   1:  PR[GP1:91,2] = PR[GP1:90,2] + -14.503;
   1:L PR[91] R[100]mm/sec CNT100;
   1:  PR[GP1:91,1] = PR[GP1:90,1] + -1.505;
   1:  PR[GP1:91,2] = PR[GP1:90,2] + -14.417;
   1:L PR[91] R[100]mm/sec CNT100;
   1:  PR[GP1:91,1] = PR[GP1:90,1] + -1.291;
   1:  PR[GP1:91,2] = PR[GP1:90,2] + -14.246;
   1:L PR[91] R[100]mm/sec CNT100;
   1:  PR[GP1:91,1] = PR[GP1:90,1] + -0.380;
   1:  PR[GP1:91,2] = PR[GP1:90,2] + -13.601;
   1:L PR[91] R[100]mm/sec CNT100;
   1:  PR[GP1:91,1] = PR[GP1:90,1] + 1.422;
   1:  PR[GP1:91,2] = PR[GP1:90,2] + -14.238;
   1:L PR[91] R[100]mm/sec CNT100;
   1:  PR[GP1:91,1] = PR[GP1:90,1] + 2.035;
   1:  PR[GP1:91,2] = PR[GP1:90,2] + -14.610;
   1:L PR[91] R[100]mm/sec CNT100;
   1:  PR[GP1:91,1] = PR[GP1:90,1] + 3.752;
   1:  PR[GP1:91,2] = PR[GP1:90,2] + -16.116;
   1:L PR[91] R[100]mm/sec CNT100;
   1:  PR[GP1:91,1] = PR[GP1:90,1] + 4.817;
   1:  PR[GP1:91,2] = PR[GP1:90,2] + -16.798;
   1:L PR[91] R[100]mm/sec CNT100;
   1:  PR[GP1:91,1] = PR[GP1:90,1] + 5.963;
   1:  PR[GP1:91,2] = PR[GP1:90,2] + -17.587;
   1:L PR[91] R[100]mm/sec CNT100;
   1:  PR[GP1:91,1] = PR[GP1:90,1] + 7.771;
   1:  PR[GP1:91,2] = PR[GP1:90,2] + -18.377;
   1:L PR[91] R[100]mm/sec CNT100;
   1:  PR[GP1:91,1] = PR[GP1:90,1] + 10.090;
   1:  PR[GP1:91,2] = PR[GP1:90,2] + -19.365;
   1:L PR[91] R[100]mm/sec CNT100;
   1:  PR[GP1:91,1] = PR[GP1:90,1] + 12.101;
   1:  PR[GP1:91,2] = PR[GP1:90,2] + -19.886;
   1:L PR[91] R[100]mm/sec CNT100;
   1:  PR[GP1:91,1] = PR[GP1:90,1] + 14.567;
   1:  PR[GP1:91,2] = PR[GP1:90,2] + -20.145;
   1:L PR[91] R[100]mm/sec CNT100;
   1:  PR[GP1:91,1] = PR[GP1:90,1] + 16.414;
   1:  PR[GP1:91,2] = PR[GP1:90,2] + -20.401;
   1:L PR[91] R[100]mm/sec CNT100;
   1:  PR[GP1:91,1] = PR[GP1:90,1] + 18.916;
   1:  PR[GP1:91,2] = PR[GP1:90,2] + -20.272;
   1:L PR[91] R[100]mm/sec CNT100;
   1:  PR[GP1:91,1] = PR[GP1:90,1] + 20.354;
   1:  PR[GP1:91,2] = PR[GP1:90,2] + -20.104;
   1:L PR[91] R[100]mm/sec CNT100;
   1:  PR[GP1:91,1] = PR[GP1:90,1] + 22.923;
   1:  PR[GP1:91,2] = PR[GP1:90,2] + -19.572;
   1:L PR[91] R[100]mm/sec CNT100;
   1:  PR[GP1:91,1] = PR[GP1:90,1] + 25.749;
   1:  PR[GP1:91,2] = PR[GP1:90,2] + -18.528;
   1:L PR[91] R[100]mm/sec CNT100;
   1:  PR[GP1:91,1] = PR[GP1:90,1] + 26.499;
   1:  PR[GP1:91,2] = PR[GP1:90,2] + -18.236;
   1:L PR[91] R[100]mm/sec CNT100;
   1:  PR[GP1:91,1] = PR[GP1:90,1] + 29.104;
   1:  PR[GP1:91,2] = PR[GP1:90,2] + -16.785;
   1:L PR[91] R[100]mm/sec CNT100;
   1:  PR[GP1:91,1] = PR[GP1:90,1] + 31.898;
   1:  PR[GP1:91,2] = PR[GP1:90,2] + -14.631;
   1:L PR[91] R[100]mm/sec CNT100;
   1:  PR[GP1:91,1] = PR[GP1:90,1] + 34.116;
   1:  PR[GP1:91,2] = PR[GP1:90,2] + -12.234;
   1:L PR[91] R[100]mm/sec CNT100;
   1:  PR[GP1:91,1] = PR[GP1:90,1] + 35.935;
   1:  PR[GP1:91,2] = PR[GP1:90,2] + -9.483;
   1:L PR[91] R[100]mm/sec CNT100;
   1:  PR[GP1:91,1] = PR[GP1:90,1] + 37.166;
   1:  PR[GP1:91,2] = PR[GP1:90,2] + -6.758;
   1:L PR[91] R[100]mm/sec CNT100;
   1:  PR[GP1:91,1] = PR[GP1:90,1] + 37.334;
   1:  PR[GP1:91,2] = PR[GP1:90,2] + -6.340;
   1:L PR[91] R[100]mm/sec CNT100;
   1:  PR[GP1:91,1] = PR[GP1:90,1] + 38.017;
   1:  PR[GP1:91,2] = PR[GP1:90,2] + -3.738;
   1:L PR[91] R[100]mm/sec CNT100;
   1:  PR[GP1:91,1] = PR[GP1:90,1] + 38.097;
   1:  PR[GP1:91,2] = PR[GP1:90,2] + -3.101;
   1:L PR[91] R[100]mm/sec CNT100;
   1:  PR[GP1:91,1] = PR[GP1:90,1] + 38.320;
   1:  PR[GP1:91,2] = PR[GP1:90,2] + -0.345;
   1:L PR[91] R[100]mm/sec CNT100;
   1:  PR[GP1:91,1] = PR[GP1:90,1] + 38.235;
   1:  PR[GP1:91,2] = PR[GP1:90,2] + 0.328;
   1:L PR[91] R[100]mm/sec CNT100;
   1:  PR[GP1:91,1] = PR[GP1:90,1] + 38.008;
   1:  PR[GP1:91,2] = PR[GP1:90,2] + 3.146;
   1:L PR[91] R[100]mm/sec CNT100;
   1:  PR[GP1:91,1] = PR[GP1:90,1] + 37.334;
   1:  PR[GP1:91,2] = PR[GP1:90,2] + 5.717;
   1:L PR[91] R[100]mm/sec CNT100;
   1:  PR[GP1:91,1] = PR[GP1:90,1] + 37.165;
   1:  PR[GP1:91,2] = PR[GP1:90,2] + 6.134;
   1:L PR[91] R[100]mm/sec CNT100;
   1:  PR[GP1:91,1] = PR[GP1:90,1] + 35.947;
   1:  PR[GP1:91,2] = PR[GP1:90,2] + 8.833;
   1:L PR[91] R[100]mm/sec CNT100;
   1:  PR[GP1:91,1] = PR[GP1:90,1] + 35.844;
   1:  PR[GP1:91,2] = PR[GP1:90,2] + 8.976;
   1:L PR[91] R[100]mm/sec CNT100;
   1:  PR[GP1:91,1] = PR[GP1:90,1] + 34.115;
   1:  PR[GP1:91,2] = PR[GP1:90,2] + 11.612;
   1:L PR[91] R[100]mm/sec CNT100;
   1:  PR[GP1:91,1] = PR[GP1:90,1] + 31.896;
   1:  PR[GP1:91,2] = PR[GP1:90,2] + 14.009;
   1:L PR[91] R[100]mm/sec CNT100;
   1:  PR[GP1:91,1] = PR[GP1:90,1] + 29.489;
   1:  PR[GP1:91,2] = PR[GP1:90,2] + 15.885;
   1:L PR[91] R[100]mm/sec CNT100;
   1:  PR[GP1:91,1] = PR[GP1:90,1] + 29.124;
   1:  PR[GP1:91,2] = PR[GP1:90,2] + 16.150;
   1:L PR[91] R[100]mm/sec CNT100;
   1:  PR[GP1:91,1] = PR[GP1:90,1] + 26.515;
   1:  PR[GP1:91,2] = PR[GP1:90,2] + 17.604;
   1:L PR[91] R[100]mm/sec CNT100;
   1:  PR[GP1:91,1] = PR[GP1:90,1] + 23.898;
   1:  PR[GP1:91,2] = PR[GP1:90,2] + 18.565;
   1:L PR[91] R[100]mm/sec CNT100;
   1:  PR[GP1:91,1] = PR[GP1:90,1] + 22.917;
   1:  PR[GP1:91,2] = PR[GP1:90,2] + 18.949;
   1:L PR[91] R[100]mm/sec CNT100;
   1:  PR[GP1:91,1] = PR[GP1:90,1] + 20.361;
   1:  PR[GP1:91,2] = PR[GP1:90,2] + 19.478;
   1:L PR[91] R[100]mm/sec CNT100;
   1:  PR[GP1:91,1] = PR[GP1:90,1] + 18.927;
   1:  PR[GP1:91,2] = PR[GP1:90,2] + 19.648;
   1:L PR[91] R[100]mm/sec CNT100;
   1:  PR[GP1:91,1] = PR[GP1:90,1] + 16.401;
   1:  PR[GP1:91,2] = PR[GP1:90,2] + 19.779;
   1:L PR[91] R[100]mm/sec CNT100;
   1:  PR[GP1:91,1] = PR[GP1:90,1] + 14.148;
   1:  PR[GP1:91,2] = PR[GP1:90,2] + 19.550;
   1:L PR[91] R[100]mm/sec CNT100;
   1:  PR[GP1:91,1] = PR[GP1:90,1] + 12.143;
   1:  PR[GP1:91,2] = PR[GP1:90,2] + 19.273;
   1:L PR[91] R[100]mm/sec CNT100;
   1:  PR[GP1:91,1] = PR[GP1:90,1] + 10.117;
   1:  PR[GP1:91,2] = PR[GP1:90,2] + 18.748;
   1:L PR[91] R[100]mm/sec CNT100;
   1:  PR[GP1:91,1] = PR[GP1:90,1] + 8.321;
   1:  PR[GP1:91,2] = PR[GP1:90,2] + 17.962;
   1:L PR[91] R[100]mm/sec CNT100;
   1:  PR[GP1:91,1] = PR[GP1:90,1] + 6.001;
   1:  PR[GP1:91,2] = PR[GP1:90,2] + 16.993;
   1:L PR[91] R[100]mm/sec CNT100;
   1:  PR[GP1:91,1] = PR[GP1:90,1] + 4.512;
   1:  PR[GP1:91,2] = PR[GP1:90,2] + 16.042;
   1:L PR[91] R[100]mm/sec CNT100;
   1:  PR[GP1:91,1] = PR[GP1:90,1] + 4.067;
   1:  PR[GP1:91,2] = PR[GP1:90,2] + 15.735;
   1:L PR[91] R[100]mm/sec CNT100;
   1:  PR[GP1:91,1] = PR[GP1:90,1] + 3.250;
   1:  PR[GP1:91,2] = PR[GP1:90,2] + 15.089;
   1:L PR[91] R[100]mm/sec CNT100;
   1:  PR[GP1:91,1] = PR[GP1:90,1] + 2.066;
   1:  PR[GP1:91,2] = PR[GP1:90,2] + 14.039;
   1:L PR[91] R[100]mm/sec CNT100;
   1:  PR[GP1:91,1] = PR[GP1:90,1] + 1.546;
   1:  PR[GP1:91,2] = PR[GP1:90,2] + 13.686;
   1:L PR[91] R[100]mm/sec CNT100;
   1:  PR[GP1:91,1] = PR[GP1:90,1] + 0.531;
   1:  PR[GP1:91,2] = PR[GP1:90,2] + 13.144;
   1:L PR[91] R[100]mm/sec CNT100;
   1:  PR[GP1:91,1] = PR[GP1:90,1] + -0.464;
   1:L PR[91] R[100]mm/sec CNT100;
   1:  PR[91] = PR[90];
   1:  PR[GP1:91,1] = PR[GP1:90,1] + -1.737;
   1:  PR[GP1:91,2] = PR[GP1:90,2] + 14.036;
   1:  PR[GP1:91,3] = PR[GP1:90,3] + 31.415;
   1:L PR[91] R[100]mm/sec CNT100;
   1:  PR[GP1:91,1] = PR[GP1:90,1] + -2.061;
   1:  PR[GP1:91,2] = PR[GP1:90,2] + 14.458;
   1:L PR[91] R[100]mm/sec CNT100;
   1:  PR[GP1:91,1] = PR[GP1:90,1] + -2.803;
   1:  PR[GP1:91,2] = PR[GP1:90,2] + 15.114;
   1:L PR[91] R[100]mm/sec CNT100;
   1:  PR[GP1:91,1] = PR[GP1:90,1] + -3.663;
   1:  PR[GP1:91,2] = PR[GP1:90,2] + 15.794;
   1:L PR[91] R[100]mm/sec CNT100;
   1:  PR[GP1:91,1] = PR[GP1:90,1] + -4.821;
   1:  PR[GP1:91,2] = PR[GP1:90,2] + 16.536;
   1:L PR[91] R[100]mm/sec CNT100;
   1:  PR[GP1:91,1] = PR[GP1:90,1] + -5.585;
   1:  PR[GP1:91,2] = PR[GP1:90,2] + 17.048;
   1:L PR[91] R[100]mm/sec CNT100;
   1:  PR[GP1:91,1] = PR[GP1:90,1] + -7.301;
   1:  PR[GP1:91,2] = PR[GP1:90,2] + 17.798;
   1:L PR[91] R[100]mm/sec CNT100;
   1:  PR[GP1:91,1] = PR[GP1:90,1] + -9.760;
   1:  PR[GP1:91,2] = PR[GP1:90,2] + 18.828;
   1:L PR[91] R[100]mm/sec CNT100;
   1:  PR[GP1:91,1] = PR[GP1:90,1] + -11.641;
   1:  PR[GP1:91,2] = PR[GP1:90,2] + 19.314;
   1:L PR[91] R[100]mm/sec CNT100;
   1:  PR[GP1:91,1] = PR[GP1:90,1] + -13.962;
   1:  PR[GP1:91,2] = PR[GP1:90,2] + 19.556;
   1:L PR[91] R[100]mm/sec CNT100;
   1:  PR[GP1:91,1] = PR[GP1:90,1] + -16.053;
   1:  PR[GP1:91,2] = PR[GP1:90,2] + 19.841;
   1:L PR[91] R[100]mm/sec CNT100;
   1:  PR[GP1:91,1] = PR[GP1:90,1] + -18.424;
   1:  PR[GP1:91,2] = PR[GP1:90,2] + 19.716;
   1:L PR[91] R[100]mm/sec CNT100;
   1:  PR[GP1:91,1] = PR[GP1:90,1] + -20.099;
   1:  PR[GP1:91,2] = PR[GP1:90,2] + 19.518;
   1:L PR[91] R[100]mm/sec CNT100;
   1:  PR[GP1:91,1] = PR[GP1:90,1] + -22.538;
   1:  PR[GP1:91,2] = PR[GP1:90,2] + 19.012;
   1:L PR[91] R[100]mm/sec CNT100;
   1:  PR[GP1:91,1] = PR[GP1:90,1] + -25.216;
   1:  PR[GP1:91,2] = PR[GP1:90,2] + 18.018;
   1:L PR[91] R[100]mm/sec CNT100;
   1:  PR[GP1:91,1] = PR[GP1:90,1] + -26.201;
   1:  PR[GP1:91,2] = PR[GP1:90,2] + 17.633;
   1:L PR[91] R[100]mm/sec CNT100;
   1:  PR[GP1:91,1] = PR[GP1:90,1] + -28.688;
   1:  PR[GP1:91,2] = PR[GP1:90,2] + 16.240;
   1:L PR[91] R[100]mm/sec CNT100;
   1:  PR[GP1:91,1] = PR[GP1:90,1] + -31.245;
   1:  PR[GP1:91,2] = PR[GP1:90,2] + 14.250;
   1:L PR[91] R[100]mm/sec CNT100;
   1:  PR[GP1:91,1] = PR[GP1:90,1] + -31.607;
   1:  PR[GP1:91,2] = PR[GP1:90,2] + 13.986;
   1:L PR[91] R[100]mm/sec CNT100;
   1:  PR[GP1:91,1] = PR[GP1:90,1] + -33.725;
   1:  PR[GP1:91,2] = PR[GP1:90,2] + 11.698;
   1:L PR[91] R[100]mm/sec CNT100;
   1:  PR[GP1:91,1] = PR[GP1:90,1] + -33.835;
   1:  PR[GP1:91,2] = PR[GP1:90,2] + 11.562;
   1:L PR[91] R[100]mm/sec CNT100;
   1:  PR[GP1:91,1] = PR[GP1:90,1] + -35.600;
   1:  PR[GP1:91,2] = PR[GP1:90,2] + 8.880;
   1:L PR[91] R[100]mm/sec CNT100;
   1:  PR[GP1:91,1] = PR[GP1:90,1] + -36.981;
   1:  PR[GP1:91,2] = PR[GP1:90,2] + 5.781;
   1:L PR[91] R[100]mm/sec CNT100;
   1:  PR[GP1:91,1] = PR[GP1:90,1] + -37.733;
   1:  PR[GP1:91,2] = PR[GP1:90,2] + 2.874;
   1:L PR[91] R[100]mm/sec CNT100;
   1:  PR[GP1:91,1] = PR[GP1:90,1] + -37.753;
   1:  PR[GP1:91,2] = PR[GP1:90,2] + 2.713;
   1:L PR[91] R[100]mm/sec CNT100;
   1:  PR[GP1:91,1] = PR[GP1:90,1] + -37.990;
   1:  PR[GP1:91,2] = PR[GP1:90,2] + -0.277;
   1:L PR[91] R[100]mm/sec CNT100;
   1:  PR[GP1:91,1] = PR[GP1:90,1] + -37.963;
   1:  PR[GP1:91,2] = PR[GP1:90,2] + -0.490;
   1:L PR[91] R[100]mm/sec CNT100;
   1:  PR[GP1:91,1] = PR[GP1:90,1] + -37.724;
   1:  PR[GP1:91,2] = PR[GP1:90,2] + -3.531;
   1:L PR[91] R[100]mm/sec CNT100;
   1:  PR[GP1:91,1] = PR[GP1:90,1] + -36.981;
   1:  PR[GP1:91,2] = PR[GP1:90,2] + -6.405;
   1:L PR[91] R[100]mm/sec CNT100;
   1:  PR[GP1:91,1] = PR[GP1:90,1] + -35.600;
   1:  PR[GP1:91,2] = PR[GP1:90,2] + -9.504;
   1:L PR[91] R[100]mm/sec CNT100;
   1:  PR[GP1:91,1] = PR[GP1:90,1] + -33.835;
   1:  PR[GP1:91,2] = PR[GP1:90,2] + -12.186;
   1:L PR[91] R[100]mm/sec CNT100;
   1:  PR[GP1:91,1] = PR[GP1:90,1] + -33.725;
   1:  PR[GP1:91,2] = PR[GP1:90,2] + -12.322;
   1:L PR[91] R[100]mm/sec CNT100;
   1:  PR[GP1:91,1] = PR[GP1:90,1] + -31.589;
   1:  PR[GP1:91,2] = PR[GP1:90,2] + -14.630;
   1:L PR[91] R[100]mm/sec CNT100;
   1:  PR[GP1:91,1] = PR[GP1:90,1] + -29.269;
   1:  PR[GP1:91,2] = PR[GP1:90,2] + -16.445;
   1:L PR[91] R[100]mm/sec CNT100;
   1:  PR[GP1:91,1] = PR[GP1:90,1] + -28.706;
   1:  PR[GP1:91,2] = PR[GP1:90,2] + -16.854;
   1:L PR[91] R[100]mm/sec CNT100;
   1:  PR[GP1:91,1] = PR[GP1:90,1] + -26.208;
   1:  PR[GP1:91,2] = PR[GP1:90,2] + -18.253;
   1:L PR[91] R[100]mm/sec CNT100;
   1:  PR[GP1:91,1] = PR[GP1:90,1] + -23.718;
   1:  PR[GP1:91,2] = PR[GP1:90,2] + -19.173;
   1:L PR[91] R[100]mm/sec CNT100;
   1:  PR[GP1:91,1] = PR[GP1:90,1] + -22.518;
   1:  PR[GP1:91,2] = PR[GP1:90,2] + -19.641;
   1:L PR[91] R[100]mm/sec CNT100;
   1:  PR[GP1:91,1] = PR[GP1:90,1] + -20.089;
   1:  PR[GP1:91,2] = PR[GP1:90,2] + -20.145;
   1:L PR[91] R[100]mm/sec CNT100;
   1:  PR[GP1:91,1] = PR[GP1:90,1] + -18.410;
   1:  PR[GP1:91,2] = PR[GP1:90,2] + -20.340;
   1:L PR[91] R[100]mm/sec CNT100;
   1:  PR[GP1:91,1] = PR[GP1:90,1] + -16.012;
   1:  PR[GP1:91,2] = PR[GP1:90,2] + -20.467;
   1:L PR[91] R[100]mm/sec CNT100;
   1:  PR[GP1:91,1] = PR[GP1:90,1] + -13.881;
   1:  PR[GP1:91,2] = PR[GP1:90,2] + -20.252;
   1:L PR[91] R[100]mm/sec CNT100;
   1:  PR[GP1:91,1] = PR[GP1:90,1] + -11.644;
   1:  PR[GP1:91,2] = PR[GP1:90,2] + -19.939;
   1:L PR[91] R[100]mm/sec CNT100;
   1:  PR[GP1:91,1] = PR[GP1:90,1] + -9.749;
   1:  PR[GP1:91,2] = PR[GP1:90,2] + -19.449;
   1:L PR[91] R[100]mm/sec CNT100;
   1:  PR[GP1:91,1] = PR[GP1:90,1] + -8.064;
   1:  PR[GP1:91,2] = PR[GP1:90,2] + -18.710;
   1:L PR[91] R[100]mm/sec CNT100;
   1:  PR[GP1:91,1] = PR[GP1:90,1] + -5.488;
   1:  PR[GP1:91,2] = PR[GP1:90,2] + -17.612;
   1:L PR[91] R[100]mm/sec CNT100;
   1:  PR[GP1:91,1] = PR[GP1:90,1] + -4.127;
   1:  PR[GP1:91,2] = PR[GP1:90,2] + -16.742;
   1:L PR[91] R[100]mm/sec CNT100;
   1:  PR[GP1:91,1] = PR[GP1:90,1] + -3.375;
   1:  PR[GP1:91,2] = PR[GP1:90,2] + -16.200;
   1:L PR[91] R[100]mm/sec CNT100;
   1:  PR[GP1:91,1] = PR[GP1:90,1] + -1.738;
   1:  PR[GP1:91,2] = PR[GP1:90,2] + -14.767;
   1:L PR[91] R[100]mm/sec CNT100;
   1:  PR[GP1:91,1] = PR[GP1:90,1] + -1.337;
   1:  PR[GP1:91,2] = PR[GP1:90,2] + -14.630;
   1:L PR[91] R[100]mm/sec CNT100;
   1:  PR[GP1:91,1] = PR[GP1:90,1] + -0.386;
   1:  PR[GP1:91,2] = PR[GP1:90,2] + -13.904;
   1:L PR[91] R[100]mm/sec CNT100;
   1:  PR[GP1:91,1] = PR[GP1:90,1] + 0.996;
   1:  PR[GP1:91,2] = PR[GP1:90,2] + -14.395;
   1:L PR[91] R[100]mm/sec CNT100;
   1:  PR[GP1:91,1] = PR[GP1:90,1] + 1.349;
   1:  PR[GP1:91,2] = PR[GP1:90,2] + -14.458;
   1:L PR[91] R[100]mm/sec CNT100;
   1:  PR[GP1:91,1] = PR[GP1:90,1] + 2.023;
   1:  PR[GP1:91,2] = PR[GP1:90,2] + -14.880;
   1:L PR[91] R[100]mm/sec CNT100;
   1:  PR[GP1:91,1] = PR[GP1:90,1] + 3.507;
   1:  PR[GP1:91,2] = PR[GP1:90,2] + -16.181;
   1:L PR[91] R[100]mm/sec CNT100;
   1:  PR[GP1:91,1] = PR[GP1:90,1] + 4.420;
   1:  PR[GP1:91,2] = PR[GP1:90,2] + -16.766;
   1:L PR[91] R[100]mm/sec CNT100;
   1:  PR[GP1:91,1] = PR[GP1:90,1] + 5.669;
   1:  PR[GP1:91,2] = PR[GP1:90,2] + -17.626;
   1:L PR[91] R[100]mm/sec CNT100;
   1:  PR[GP1:91,1] = PR[GP1:90,1] + 7.347;
   1:  PR[GP1:91,2] = PR[GP1:90,2] + -18.359;
   1:L PR[91] R[100]mm/sec CNT100;
   1:  PR[GP1:91,1] = PR[GP1:90,1] + 9.893;
   1:  PR[GP1:91,2] = PR[GP1:90,2] + -19.443;
   1:L PR[91] R[100]mm/sec CNT100;
   1:  PR[GP1:91,1] = PR[GP1:90,1] + 11.774;
   1:  PR[GP1:91,2] = PR[GP1:90,2] + -19.931;
   1:L PR[91] R[100]mm/sec CNT100;
   1:  PR[GP1:91,1] = PR[GP1:90,1] + 14.091;
   1:  PR[GP1:91,2] = PR[GP1:90,2] + -20.174;
   1:L PR[91] R[100]mm/sec CNT100;
   1:  PR[GP1:91,1] = PR[GP1:90,1] + 16.188;
   1:  PR[GP1:91,2] = PR[GP1:90,2] + -20.465;
   1:L PR[91] R[100]mm/sec CNT100;
   1:  PR[GP1:91,1] = PR[GP1:90,1] + 18.547;
   1:  PR[GP1:91,2] = PR[GP1:90,2] + -20.343;
   1:L PR[91] R[100]mm/sec CNT100;
   1:  PR[GP1:91,1] = PR[GP1:90,1] + 20.228;
   1:  PR[GP1:91,2] = PR[GP1:90,2] + -20.147;
   1:L PR[91] R[100]mm/sec CNT100;
   1:  PR[GP1:91,1] = PR[GP1:90,1] + 22.665;
   1:  PR[GP1:91,2] = PR[GP1:90,2] + -19.643;
   1:L PR[91] R[100]mm/sec CNT100;
   1:  PR[GP1:91,1] = PR[GP1:90,1] + 25.348;
   1:  PR[GP1:91,2] = PR[GP1:90,2] + -18.652;
   1:L PR[91] R[100]mm/sec CNT100;
   1:  PR[GP1:91,1] = PR[GP1:90,1] + 26.337;
   1:  PR[GP1:91,2] = PR[GP1:90,2] + -18.267;
   1:L PR[91] R[100]mm/sec CNT100;
   1:  PR[GP1:91,1] = PR[GP1:90,1] + 28.815;
   1:  PR[GP1:91,2] = PR[GP1:90,2] + -16.886;
   1:L PR[91] R[100]mm/sec CNT100;
   1:  PR[GP1:91,1] = PR[GP1:90,1] + 31.351;
   1:  PR[GP1:91,2] = PR[GP1:90,2] + -14.921;
   1:L PR[91] R[100]mm/sec CNT100;
   1:  PR[GP1:91,1] = PR[GP1:90,1] + 31.718;
   1:  PR[GP1:91,2] = PR[GP1:90,2] + -14.655;
   1:L PR[91] R[100]mm/sec CNT100;
   1:  PR[GP1:91,1] = PR[GP1:90,1] + 33.841;
   1:  PR[GP1:91,2] = PR[GP1:90,2] + -12.364;
   1:L PR[91] R[100]mm/sec CNT100;
   1:  PR[GP1:91,1] = PR[GP1:90,1] + 33.955;
   1:  PR[GP1:91,2] = PR[GP1:90,2] + -12.223;
   1:L PR[91] R[100]mm/sec CNT100;
   1:  PR[GP1:91,1] = PR[GP1:90,1] + 35.744;
   1:  PR[GP1:91,2] = PR[GP1:90,2] + -9.519;
   1:L PR[91] R[100]mm/sec CNT100;
   1:  PR[GP1:91,1] = PR[GP1:90,1] + 36.572;
   1:  PR[GP1:91,2] = PR[GP1:90,2] + -7.697;
   1:L PR[91] R[100]mm/sec CNT100;
   1:  PR[GP1:91,1] = PR[GP1:90,1] + 37.122;
   1:  PR[GP1:91,2] = PR[GP1:90,2] + -6.469;
   1:L PR[91] R[100]mm/sec CNT100;
   1:  PR[GP1:91,1] = PR[GP1:90,1] + 37.876;
   1:  PR[GP1:91,2] = PR[GP1:90,2] + -3.591;
   1:L PR[91] R[100]mm/sec CNT100;
   1:  PR[GP1:91,1] = PR[GP1:90,1] + 37.896;
   1:  PR[GP1:91,2] = PR[GP1:90,2] + -3.433;
   1:L PR[91] R[100]mm/sec CNT100;
   1:  PR[GP1:91,1] = PR[GP1:90,1] + 38.147;
   1:  PR[GP1:91,2] = PR[GP1:90,2] + -0.345;
   1:L PR[91] R[100]mm/sec CNT100;
   1:  PR[GP1:91,1] = PR[GP1:90,1] + 38.120;
   1:  PR[GP1:91,2] = PR[GP1:90,2] + -0.134;
   1:L PR[91] R[100]mm/sec CNT100;
   1:  PR[GP1:91,1] = PR[GP1:90,1] + 37.868;
   1:  PR[GP1:91,2] = PR[GP1:90,2] + 2.999;
   1:L PR[91] R[100]mm/sec CNT100;
   1:  PR[GP1:91,1] = PR[GP1:90,1] + 37.122;
   1:  PR[GP1:91,2] = PR[GP1:90,2] + 5.843;
   1:L PR[91] R[100]mm/sec CNT100;
   1:  PR[GP1:91,1] = PR[GP1:90,1] + 35.744;
   1:  PR[GP1:91,2] = PR[GP1:90,2] + 8.896;
   1:L PR[91] R[100]mm/sec CNT100;
   1:  PR[GP1:91,1] = PR[GP1:90,1] + 33.955;
   1:  PR[GP1:91,2] = PR[GP1:90,2] + 11.599;
   1:L PR[91] R[100]mm/sec CNT100;
   1:  PR[GP1:91,1] = PR[GP1:90,1] + 33.842;
   1:  PR[GP1:91,2] = PR[GP1:90,2] + 11.740;
   1:L PR[91] R[100]mm/sec CNT100;
   1:  PR[GP1:91,1] = PR[GP1:90,1] + 31.702;
   1:  PR[GP1:91,2] = PR[GP1:90,2] + 14.047;
   1:L PR[91] R[100]mm/sec CNT100;
   1:  PR[GP1:91,1] = PR[GP1:90,1] + 29.402;
   1:  PR[GP1:91,2] = PR[GP1:90,2] + 15.840;
   1:L PR[91] R[100]mm/sec CNT100;
   1:  PR[GP1:91,1] = PR[GP1:90,1] + 28.838;
   1:  PR[GP1:91,2] = PR[GP1:90,2] + 16.249;
   1:L PR[91] R[100]mm/sec CNT100;
   1:  PR[GP1:91,1] = PR[GP1:90,1] + 26.354;
   1:  PR[GP1:91,2] = PR[GP1:90,2] + 17.634;
   1:L PR[91] R[100]mm/sec CNT100;
   1:  PR[GP1:91,1] = PR[GP1:90,1] + 23.860;
   1:  PR[GP1:91,2] = PR[GP1:90,2] + 18.550;
   1:L PR[91] R[100]mm/sec CNT100;
   1:  PR[GP1:91,1] = PR[GP1:90,1] + 22.660;
   1:  PR[GP1:91,2] = PR[GP1:90,2] + 19.019;
   1:L PR[91] R[100]mm/sec CNT100;
   1:  PR[GP1:91,1] = PR[GP1:90,1] + 20.237;
   1:  PR[GP1:91,2] = PR[GP1:90,2] + 19.521;
   1:L PR[91] R[100]mm/sec CNT100;
   1:  PR[GP1:91,1] = PR[GP1:90,1] + 18.561;
   1:  PR[GP1:91,2] = PR[GP1:90,2] + 19.719;
   1:L PR[91] R[100]mm/sec CNT100;
   1:  PR[GP1:91,1] = PR[GP1:90,1] + 16.177;
   1:  PR[GP1:91,2] = PR[GP1:90,2] + 19.843;
   1:L PR[91] R[100]mm/sec CNT100;
   1:  PR[GP1:91,1] = PR[GP1:90,1] + 14.051;
   1:  PR[GP1:91,2] = PR[GP1:90,2] + 19.627;
   1:L PR[91] R[100]mm/sec CNT100;
   1:  PR[GP1:91,1] = PR[GP1:90,1] + 11.818;
   1:  PR[GP1:91,2] = PR[GP1:90,2] + 19.319;
   1:L PR[91] R[100]mm/sec CNT100;
   1:  PR[GP1:91,1] = PR[GP1:90,1] + 9.921;
   1:  PR[GP1:91,2] = PR[GP1:90,2] + 18.827;
   1:L PR[91] R[100]mm/sec CNT100;
   1:  PR[GP1:91,1] = PR[GP1:90,1] + 8.235;
   1:  PR[GP1:91,2] = PR[GP1:90,2] + 18.089;
   1:L PR[91] R[100]mm/sec CNT100;
   1:  PR[GP1:91,1] = PR[GP1:90,1] + 5.713;
   1:  PR[GP1:91,2] = PR[GP1:90,2] + 17.035;
   1:L PR[91] R[100]mm/sec CNT100;
   1:  PR[GP1:91,1] = PR[GP1:90,1] + 4.329;
   1:  PR[GP1:91,2] = PR[GP1:90,2] + 16.152;
   1:L PR[91] R[100]mm/sec CNT100;
   1:  PR[GP1:91,1] = PR[GP1:90,1] + 3.846;
   1:  PR[GP1:91,2] = PR[GP1:90,2] + 15.818;
   1:L PR[91] R[100]mm/sec CNT100;
   1:  PR[GP1:91,1] = PR[GP1:90,1] + 2.962;
   1:  PR[GP1:91,2] = PR[GP1:90,2] + 15.119;
   1:L PR[91] R[100]mm/sec CNT100;
   1:  PR[GP1:91,1] = PR[GP1:90,1] + 2.045;
   1:  PR[GP1:91,2] = PR[GP1:90,2] + 14.306;
   1:L PR[91] R[100]mm/sec CNT100;
   1:  PR[GP1:91,1] = PR[GP1:90,1] + 1.786;
   1:  PR[GP1:91,2] = PR[GP1:90,2] + 14.131;
   1:L PR[91] R[100]mm/sec CNT100;
   1:  PR[GP1:91,1] = PR[GP1:90,1] + 1.502;
   1:  PR[GP1:91,2] = PR[GP1:90,2] + 13.855;
   1:L PR[91] R[100]mm/sec CNT100;
   1:  PR[GP1:91,1] = PR[GP1:90,1] + 1.098;
   1:  PR[GP1:91,2] = PR[GP1:90,2] + 13.786;
   1:L PR[91] R[100]mm/sec CNT100;
   1:  PR[GP1:91,1] = PR[GP1:90,1] + 0.499;
   1:  PR[GP1:91,2] = PR[GP1:90,2] + 13.458;
   1:L PR[91] R[100]mm/sec CNT100;
   1:  PR[GP1:91,1] = PR[GP1:90,1] + -0.440;
   1:L PR[91] R[100]mm/sec CNT100;
   1:  PR[91] = PR[90];
   1:  PR[GP1:91,1] = PR[GP1:90,1] + -1.776;
   1:  PR[GP1:91,2] = PR[GP1:90,2] + 14.379;
   1:  PR[GP1:91,3] = PR[GP1:90,3] + 32.025;
   1:L PR[91] R[100]mm/sec CNT100;
   1:  PR[GP1:91,1] = PR[GP1:90,1] + -2.043;
   1:  PR[GP1:91,2] = PR[GP1:90,2] + 14.727;
   1:L PR[91] R[100]mm/sec CNT100;
   1:  PR[GP1:91,1] = PR[GP1:90,1] + -2.516;
   1:  PR[GP1:91,2] = PR[GP1:90,2] + 15.145;
   1:L PR[91] R[100]mm/sec CNT100;
   1:  PR[GP1:91,1] = PR[GP1:90,1] + -3.443;
   1:  PR[GP1:91,2] = PR[GP1:90,2] + 15.878;
   1:L PR[91] R[100]mm/sec CNT100;
   1:  PR[GP1:91,1] = PR[GP1:90,1] + -4.468;
   1:  PR[GP1:91,2] = PR[GP1:90,2] + 16.534;
   1:L PR[91] R[100]mm/sec CNT100;
   1:  PR[GP1:91,1] = PR[GP1:90,1] + -5.298;
   1:  PR[GP1:91,2] = PR[GP1:90,2] + 17.091;
   1:L PR[91] R[100]mm/sec CNT100;
   1:  PR[GP1:91,1] = PR[GP1:90,1] + -6.886;
   1:  PR[GP1:91,2] = PR[GP1:90,2] + 17.785;
   1:L PR[91] R[100]mm/sec CNT100;
   1:  PR[GP1:91,1] = PR[GP1:90,1] + -9.564;
   1:  PR[GP1:91,2] = PR[GP1:90,2] + 18.907;
   1:L PR[91] R[100]mm/sec CNT100;
   1:  PR[GP1:91,1] = PR[GP1:90,1] + -11.316;
   1:  PR[GP1:91,2] = PR[GP1:90,2] + 19.360;
   1:L PR[91] R[100]mm/sec CNT100;
   1:  PR[GP1:91,1] = PR[GP1:90,1] + -13.488;
   1:  PR[GP1:91,2] = PR[GP1:90,2] + 19.586;
   1:L PR[91] R[100]mm/sec CNT100;
   1:  PR[GP1:91,1] = PR[GP1:90,1] + -15.829;
   1:  PR[GP1:91,2] = PR[GP1:90,2] + 19.905;
   1:L PR[91] R[100]mm/sec CNT100;
   1:  PR[GP1:91,1] = PR[GP1:90,1] + -18.057;
   1:  PR[GP1:91,2] = PR[GP1:90,2] + 19.788;
   1:L PR[91] R[100]mm/sec CNT100;
   1:  PR[GP1:91,1] = PR[GP1:90,1] + -19.974;
   1:  PR[GP1:91,2] = PR[GP1:90,2] + 19.561;
   1:L PR[91] R[100]mm/sec CNT100;
   1:  PR[GP1:91,1] = PR[GP1:90,1] + -22.280;
   1:  PR[GP1:91,2] = PR[GP1:90,2] + 19.083;
   1:L PR[91] R[100]mm/sec CNT100;
   1:  PR[GP1:91,1] = PR[GP1:90,1] + -24.815;
   1:  PR[GP1:91,2] = PR[GP1:90,2] + 18.142;
   1:L PR[91] R[100]mm/sec CNT100;
   1:  PR[GP1:91,1] = PR[GP1:90,1] + -26.039;
   1:  PR[GP1:91,2] = PR[GP1:90,2] + 17.663;
   1:L PR[91] R[100]mm/sec CNT100;
   1:  PR[GP1:91,1] = PR[GP1:90,1] + -28.400;
   1:  PR[GP1:91,2] = PR[GP1:90,2] + 16.340;
   1:L PR[91] R[100]mm/sec CNT100;
   1:  PR[GP1:91,1] = PR[GP1:90,1] + -30.833;
   1:  PR[GP1:91,2] = PR[GP1:90,2] + 14.447;
   1:L PR[91] R[100]mm/sec CNT100;
   1:  PR[GP1:91,1] = PR[GP1:90,1] + -31.411;
   1:  PR[GP1:91,2] = PR[GP1:90,2] + 14.026;
   1:L PR[91] R[100]mm/sec CNT100;
   1:  PR[GP1:91,1] = PR[GP1:90,1] + -33.429;
   1:  PR[GP1:91,2] = PR[GP1:90,2] + 11.846;
   1:L PR[91] R[100]mm/sec CNT100;
   1:  PR[GP1:91,1] = PR[GP1:90,1] + -33.699;
   1:  PR[GP1:91,2] = PR[GP1:90,2] + 11.511;
   1:L PR[91] R[100]mm/sec CNT100;
   1:  PR[GP1:91,1] = PR[GP1:90,1] + -35.386;
   1:  PR[GP1:91,2] = PR[GP1:90,2] + 8.948;
   1:L PR[91] R[100]mm/sec CNT100;
   1:  PR[GP1:91,1] = PR[GP1:90,1] + -36.796;
   1:  PR[GP1:91,2] = PR[GP1:90,2] + 5.798;
   1:L PR[91] R[100]mm/sec CNT100;
   1:  PR[GP1:91,1] = PR[GP1:90,1] + -37.557;
   1:  PR[GP1:91,2] = PR[GP1:90,2] + 2.858;
   1:L PR[91] R[100]mm/sec CNT100;
   1:  PR[GP1:91,1] = PR[GP1:90,1] + -37.815;
   1:  PR[GP1:91,2] = PR[GP1:90,2] + -0.313;
   1:L PR[91] R[100]mm/sec CNT100;
   1:  PR[GP1:91,1] = PR[GP1:90,1] + -37.566;
   1:  PR[GP1:91,2] = PR[GP1:90,2] + -3.449;
   1:L PR[91] R[100]mm/sec CNT100;
   1:  PR[GP1:91,1] = PR[GP1:90,1] + -36.796;
   1:  PR[GP1:91,2] = PR[GP1:90,2] + -6.422;
   1:L PR[91] R[100]mm/sec CNT100;
   1:  PR[GP1:91,1] = PR[GP1:90,1] + -35.470;
   1:  PR[GP1:91,2] = PR[GP1:90,2] + -9.377;
   1:L PR[91] R[100]mm/sec CNT100;
   1:  PR[GP1:91,1] = PR[GP1:90,1] + -35.382;
   1:  PR[GP1:91,2] = PR[GP1:90,2] + -9.577;
   1:L PR[91] R[100]mm/sec CNT100;
   1:  PR[GP1:91,1] = PR[GP1:90,1] + -33.699;
   1:  PR[GP1:91,2] = PR[GP1:90,2] + -12.135;
   1:L PR[91] R[100]mm/sec CNT100;
   1:  PR[GP1:91,1] = PR[GP1:90,1] + -33.428;
   1:  PR[GP1:91,2] = PR[GP1:90,2] + -12.471;
   1:L PR[91] R[100]mm/sec CNT100;
   1:  PR[GP1:91,1] = PR[GP1:90,1] + -31.392;
   1:  PR[GP1:91,2] = PR[GP1:90,2] + -14.670;
   1:L PR[91] R[100]mm/sec CNT100;
   1:  PR[GP1:91,1] = PR[GP1:90,1] + -29.180;
   1:  PR[GP1:91,2] = PR[GP1:90,2] + -16.402;
   1:L PR[91] R[100]mm/sec CNT100;
   1:  PR[GP1:91,1] = PR[GP1:90,1] + -28.417;
   1:  PR[GP1:91,2] = PR[GP1:90,2] + -16.955;
   1:L PR[91] R[100]mm/sec CNT100;
   1:  PR[GP1:91,1] = PR[GP1:90,1] + -26.045;
   1:  PR[GP1:91,2] = PR[GP1:90,2] + -18.284;
   1:L PR[91] R[100]mm/sec CNT100;
   1:  PR[GP1:91,1] = PR[GP1:90,1] + -23.677;
   1:  PR[GP1:91,2] = PR[GP1:90,2] + -19.158;
   1:L PR[91] R[100]mm/sec CNT100;
   1:  PR[GP1:91,1] = PR[GP1:90,1] + -22.258;
   1:  PR[GP1:91,2] = PR[GP1:90,2] + -19.712;
   1:L PR[91] R[100]mm/sec CNT100;
   1:  PR[GP1:91,1] = PR[GP1:90,1] + -19.963;
   1:  PR[GP1:91,2] = PR[GP1:90,2] + -20.188;
   1:L PR[91] R[100]mm/sec CNT100;
   1:  PR[GP1:91,1] = PR[GP1:90,1] + -18.041;
   1:  PR[GP1:91,2] = PR[GP1:90,2] + -20.412;
   1:L PR[91] R[100]mm/sec CNT100;
   1:  PR[GP1:91,1] = PR[GP1:90,1] + -15.786;
   1:  PR[GP1:91,2] = PR[GP1:90,2] + -20.531;
   1:L PR[91] R[100]mm/sec CNT100;
   1:  PR[GP1:91,1] = PR[GP1:90,1] + -13.783;
   1:  PR[GP1:91,2] = PR[GP1:90,2] + -20.329;
   1:L PR[91] R[100]mm/sec CNT100;
   1:  PR[GP1:91,1] = PR[GP1:90,1] + -11.317;
   1:  PR[GP1:91,2] = PR[GP1:90,2] + -19.984;
   1:L PR[91] R[100]mm/sec CNT100;
   1:  PR[GP1:91,1] = PR[GP1:90,1] + -9.551;
   1:  PR[GP1:91,2] = PR[GP1:90,2] + -19.527;
   1:L PR[91] R[100]mm/sec CNT100;
   1:  PR[GP1:91,1] = PR[GP1:90,1] + -7.977;
   1:  PR[GP1:91,2] = PR[GP1:90,2] + -18.837;
   1:L PR[91] R[100]mm/sec CNT100;
   1:  PR[GP1:91,1] = PR[GP1:90,1] + -5.195;
   1:  PR[GP1:91,2] = PR[GP1:90,2] + -17.651;
   1:L PR[91] R[100]mm/sec CNT100;
   1:  PR[GP1:91,1] = PR[GP1:90,1] + -3.942;
   1:  PR[GP1:91,2] = PR[GP1:90,2] + -16.850;
   1:L PR[91] R[100]mm/sec CNT100;
   1:  PR[GP1:91,1] = PR[GP1:90,1] + -3.131;
   1:  PR[GP1:91,2] = PR[GP1:90,2] + -16.265;
   1:L PR[91] R[100]mm/sec CNT100;
   1:  PR[GP1:91,1] = PR[GP1:90,1] + -1.721;
   1:  PR[GP1:91,2] = PR[GP1:90,2] + -15.030;
   1:L PR[91] R[100]mm/sec CNT100;
   1:  PR[GP1:91,1] = PR[GP1:90,1] + -1.186;
   1:  PR[GP1:91,2] = PR[GP1:90,2] + -14.848;
   1:L PR[91] R[100]mm/sec CNT100;
   1:  PR[GP1:91,1] = PR[GP1:90,1] + -0.361;
   1:  PR[GP1:91,2] = PR[GP1:90,2] + -14.219;
   1:L PR[91] R[100]mm/sec CNT100;
   1:  PR[GP1:91,1] = PR[GP1:90,1] + 0.835;
   1:  PR[GP1:91,2] = PR[GP1:90,2] + -14.644;
   1:L PR[91] R[100]mm/sec CNT100;
   1:  PR[GP1:91,1] = PR[GP1:90,1] + 1.381;
   1:  PR[GP1:91,2] = PR[GP1:90,2] + -14.742;
   1:L PR[91] R[100]mm/sec CNT100;
   1:  PR[GP1:91,1] = PR[GP1:90,1] + 2.014;
   1:  PR[GP1:91,2] = PR[GP1:90,2] + -15.151;
   1:L PR[91] R[100]mm/sec CNT100;
   1:  PR[GP1:91,1] = PR[GP1:90,1] + 3.262;
   1:  PR[GP1:91,2] = PR[GP1:90,2] + -16.245;
   1:L PR[91] R[100]mm/sec CNT100;
   1:  PR[GP1:91,1] = PR[GP1:90,1] + 4.033;
   1:  PR[GP1:91,2] = PR[GP1:90,2] + -16.740;
   1:L PR[91] R[100]mm/sec CNT100;
   1:  PR[GP1:91,1] = PR[GP1:90,1] + 4.585;
   1:  PR[GP1:91,2] = PR[GP1:90,2] + -17.133;
   1:L PR[91] R[100]mm/sec CNT100;
   1:  PR[GP1:91,1] = PR[GP1:90,1] + 5.370;
   1:  PR[GP1:91,2] = PR[GP1:90,2] + -17.662;
   1:L PR[91] R[100]mm/sec CNT100;
   1:  PR[GP1:91,1] = PR[GP1:90,1] + 6.923;
   1:  PR[GP1:91,2] = PR[GP1:90,2] + -18.340;
   1:L PR[91] R[100]mm/sec CNT100;
   1:  PR[GP1:91,1] = PR[GP1:90,1] + 9.695;
   1:  PR[GP1:91,2] = PR[GP1:90,2] + -19.522;
   1:L PR[91] R[100]mm/sec CNT100;
   1:  PR[GP1:91,1] = PR[GP1:90,1] + 11.447;
   1:  PR[GP1:91,2] = PR[GP1:90,2] + -19.976;
   1:L PR[91] R[100]mm/sec CNT100;
   1:  PR[GP1:91,1] = PR[GP1:90,1] + 13.616;
   1:  PR[GP1:91,2] = PR[GP1:90,2] + -20.203;
   1:L PR[91] R[100]mm/sec CNT100;
   1:  PR[GP1:91,1] = PR[GP1:90,1] + 15.963;
   1:  PR[GP1:91,2] = PR[GP1:90,2] + -20.529;
   1:L PR[91] R[100]mm/sec CNT100;
   1:  PR[GP1:91,1] = PR[GP1:90,1] + 18.179;
   1:  PR[GP1:91,2] = PR[GP1:90,2] + -20.414;
   1:L PR[91] R[100]mm/sec CNT100;
   1:  PR[GP1:91,1] = PR[GP1:90,1] + 20.102;
   1:  PR[GP1:91,2] = PR[GP1:90,2] + -20.190;
   1:L PR[91] R[100]mm/sec CNT100;
   1:  PR[GP1:91,1] = PR[GP1:90,1] + 22.406;
   1:  PR[GP1:91,2] = PR[GP1:90,2] + -19.714;
   1:L PR[91] R[100]mm/sec CNT100;
   1:  PR[GP1:91,1] = PR[GP1:90,1] + 24.945;
   1:  PR[GP1:91,2] = PR[GP1:90,2] + -18.775;
   1:L PR[91] R[100]mm/sec CNT100;
   1:  PR[GP1:91,1] = PR[GP1:90,1] + 26.175;
   1:  PR[GP1:91,2] = PR[GP1:90,2] + -18.297;
   1:L PR[91] R[100]mm/sec CNT100;
   1:  PR[GP1:91,1] = PR[GP1:90,1] + 28.527;
   1:  PR[GP1:91,2] = PR[GP1:90,2] + -16.987;
   1:L PR[91] R[100]mm/sec CNT100;
   1:  PR[GP1:91,1] = PR[GP1:90,1] + 30.940;
   1:  PR[GP1:91,2] = PR[GP1:90,2] + -15.117;
   1:L PR[91] R[100]mm/sec CNT100;
   1:  PR[GP1:91,1] = PR[GP1:90,1] + 31.523;
   1:  PR[GP1:91,2] = PR[GP1:90,2] + -14.693;
   1:L PR[91] R[100]mm/sec CNT100;
   1:  PR[GP1:91,1] = PR[GP1:90,1] + 33.546;
   1:  PR[GP1:91,2] = PR[GP1:90,2] + -12.511;
   1:L PR[91] R[100]mm/sec CNT100;
   1:  PR[GP1:91,1] = PR[GP1:90,1] + 33.820;
   1:  PR[GP1:91,2] = PR[GP1:90,2] + -12.171;
   1:L PR[91] R[100]mm/sec CNT100;
   1:  PR[GP1:91,1] = PR[GP1:90,1] + 35.530;
   1:  PR[GP1:91,2] = PR[GP1:90,2] + -9.588;
   1:L PR[91] R[100]mm/sec CNT100;
   1:  PR[GP1:91,1] = PR[GP1:90,1] + 36.906;
   1:  PR[GP1:91,2] = PR[GP1:90,2] + -6.556;
   1:L PR[91] R[100]mm/sec CNT100;
   1:  PR[GP1:91,1] = PR[GP1:90,1] + 36.935;
   1:  PR[GP1:91,2] = PR[GP1:90,2] + -6.490;
   1:L PR[91] R[100]mm/sec CNT100;
   1:  PR[GP1:91,1] = PR[GP1:90,1] + 37.700;
   1:  PR[GP1:91,2] = PR[GP1:90,2] + -3.579;
   1:L PR[91] R[100]mm/sec CNT100;
   1:  PR[GP1:91,1] = PR[GP1:90,1] + 37.972;
   1:  PR[GP1:91,2] = PR[GP1:90,2] + -0.312;
   1:L PR[91] R[100]mm/sec CNT100;
   1:  PR[GP1:91,1] = PR[GP1:90,1] + 37.700;
   1:  PR[GP1:91,2] = PR[GP1:90,2] + 2.954;
   1:L PR[91] R[100]mm/sec CNT100;
   1:  PR[GP1:91,1] = PR[GP1:90,1] + 36.937;
   1:  PR[GP1:91,2] = PR[GP1:90,2] + 5.858;
   1:L PR[91] R[100]mm/sec CNT100;
   1:  PR[GP1:91,1] = PR[GP1:90,1] + 35.530;
   1:  PR[GP1:91,2] = PR[GP1:90,2] + 8.963;
   1:L PR[91] R[100]mm/sec CNT100;
   1:  PR[GP1:91,1] = PR[GP1:90,1] + 33.821;
   1:  PR[GP1:91,2] = PR[GP1:90,2] + 11.546;
   1:L PR[91] R[100]mm/sec CNT100;
   1:  PR[GP1:91,1] = PR[GP1:90,1] + 33.547;
   1:  PR[GP1:91,2] = PR[GP1:90,2] + 11.886;
   1:L PR[91] R[100]mm/sec CNT100;
   1:  PR[GP1:91,1] = PR[GP1:90,1] + 31.508;
   1:  PR[GP1:91,2] = PR[GP1:90,2] + 14.085;
   1:L PR[91] R[100]mm/sec CNT100;
   1:  PR[GP1:91,1] = PR[GP1:90,1] + 29.314;
   1:  PR[GP1:91,2] = PR[GP1:90,2] + 15.795;
   1:L PR[91] R[100]mm/sec CNT100;
   1:  PR[GP1:91,1] = PR[GP1:90,1] + 28.552;
   1:  PR[GP1:91,2] = PR[GP1:90,2] + 16.349;
   1:L PR[91] R[100]mm/sec CNT100;
   1:  PR[GP1:91,1] = PR[GP1:90,1] + 26.193;
   1:  PR[GP1:91,2] = PR[GP1:90,2] + 17.663;
   1:L PR[91] R[100]mm/sec CNT100;
   1:  PR[GP1:91,1] = PR[GP1:90,1] + 23.821;
   1:  PR[GP1:91,2] = PR[GP1:90,2] + 18.535;
   1:L PR[91] R[100]mm/sec CNT100;
   1:  PR[GP1:91,1] = PR[GP1:90,1] + 22.403;
   1:  PR[GP1:91,2] = PR[GP1:90,2] + 19.090;
   1:L PR[91] R[100]mm/sec CNT100;
   1:  PR[GP1:91,1] = PR[GP1:90,1] + 20.113;
   1:  PR[GP1:91,2] = PR[GP1:90,2] + 19.564;
   1:L PR[91] R[100]mm/sec CNT100;
   1:  PR[GP1:91,1] = PR[GP1:90,1] + 18.194;
   1:  PR[GP1:91,2] = PR[GP1:90,2] + 19.791;
   1:L PR[91] R[100]mm/sec CNT100;
   1:  PR[GP1:91,1] = PR[GP1:90,1] + 15.953;
   1:  PR[GP1:91,2] = PR[GP1:90,2] + 19.907;
   1:L PR[91] R[100]mm/sec CNT100;
   1:  PR[GP1:91,1] = PR[GP1:90,1] + 13.954;
   1:  PR[GP1:91,2] = PR[GP1:90,2] + 19.704;
   1:L PR[91] R[100]mm/sec CNT100;
   1:  PR[GP1:91,1] = PR[GP1:90,1] + 11.493;
   1:  PR[GP1:91,2] = PR[GP1:90,2] + 19.364;
   1:L PR[91] R[100]mm/sec CNT100;
   1:  PR[GP1:91,1] = PR[GP1:90,1] + 9.726;
   1:  PR[GP1:91,2] = PR[GP1:90,2] + 18.906;
   1:L PR[91] R[100]mm/sec CNT100;
   1:  PR[GP1:91,1] = PR[GP1:90,1] + 8.150;
   1:  PR[GP1:91,2] = PR[GP1:90,2] + 18.216;
   1:L PR[91] R[100]mm/sec CNT100;
   1:  PR[GP1:91,1] = PR[GP1:90,1] + 5.426;
   1:  PR[GP1:91,2] = PR[GP1:90,2] + 17.078;
   1:L PR[91] R[100]mm/sec CNT100;
   1:  PR[GP1:91,1] = PR[GP1:90,1] + 4.147;
   1:  PR[GP1:91,2] = PR[GP1:90,2] + 16.261;
   1:L PR[91] R[100]mm/sec CNT100;
   1:  PR[GP1:91,1] = PR[GP1:90,1] + 3.625;
   1:  PR[GP1:91,2] = PR[GP1:90,2] + 15.901;
   1:L PR[91] R[100]mm/sec CNT100;
   1:  PR[GP1:91,1] = PR[GP1:90,1] + 2.675;
   1:  PR[GP1:91,2] = PR[GP1:90,2] + 15.149;
   1:L PR[91] R[100]mm/sec CNT100;
   1:  PR[GP1:91,1] = PR[GP1:90,1] + 2.026;
   1:  PR[GP1:91,2] = PR[GP1:90,2] + 14.575;
   1:L PR[91] R[100]mm/sec CNT100;
   1:  PR[GP1:91,1] = PR[GP1:90,1] + 1.855;
   1:  PR[GP1:91,2] = PR[GP1:90,2] + 14.459;
   1:L PR[91] R[100]mm/sec CNT100;
   1:  PR[GP1:91,1] = PR[GP1:90,1] + 1.521;
   1:  PR[GP1:91,2] = PR[GP1:90,2] + 14.135;
   1:L PR[91] R[100]mm/sec CNT100;
   1:  PR[GP1:91,1] = PR[GP1:90,1] + 0.938;
   1:  PR[GP1:91,2] = PR[GP1:90,2] + 14.036;
   1:L PR[91] R[100]mm/sec CNT100;
   1:  PR[GP1:91,1] = PR[GP1:90,1] + 0.459;
   1:  PR[GP1:91,2] = PR[GP1:90,2] + 13.773;
   1:L PR[91] R[100]mm/sec CNT100;
   1:  PR[GP1:91,1] = PR[GP1:90,1] + -0.415;
   1:L PR[91] R[100]mm/sec CNT100;
   1:  PR[91] = PR[90];
   1:  PR[GP1:91,1] = PR[GP1:90,1] + -1.816;
   1:  PR[GP1:91,2] = PR[GP1:90,2] + 14.722;
   1:  PR[GP1:91,3] = PR[GP1:90,3] + 32.635;
   1:L PR[91] R[100]mm/sec CNT100;
   1:  PR[GP1:91,1] = PR[GP1:90,1] + -2.026;
   1:  PR[GP1:91,2] = PR[GP1:90,2] + 14.996;
   1:L PR[91] R[100]mm/sec CNT100;
   1:  PR[GP1:91,1] = PR[GP1:90,1] + -2.230;
   1:  PR[GP1:91,2] = PR[GP1:90,2] + 15.176;
   1:L PR[91] R[100]mm/sec CNT100;
   1:  PR[GP1:91,1] = PR[GP1:90,1] + -3.224;
   1:  PR[GP1:91,2] = PR[GP1:90,2] + 15.962;
   1:L PR[91] R[100]mm/sec CNT100;
   1:  PR[GP1:91,1] = PR[GP1:90,1] + -4.115;
   1:  PR[GP1:91,2] = PR[GP1:90,2] + 16.533;
   1:L PR[91] R[100]mm/sec CNT100;
   1:  PR[GP1:91,1] = PR[GP1:90,1] + -5.011;
   1:  PR[GP1:91,2] = PR[GP1:90,2] + 17.133;
   1:L PR[91] R[100]mm/sec CNT100;
   1:  PR[GP1:91,1] = PR[GP1:90,1] + -6.471;
   1:  PR[GP1:91,2] = PR[GP1:90,2] + 17.771;
   1:L PR[91] R[100]mm/sec CNT100;
   1:  PR[GP1:91,1] = PR[GP1:90,1] + -9.368;
   1:  PR[GP1:91,2] = PR[GP1:90,2] + 18.986;
   1:L PR[91] R[100]mm/sec CNT100;
   1:  PR[GP1:91,1] = PR[GP1:90,1] + -10.991;
   1:  PR[GP1:91,2] = PR[GP1:90,2] + 19.405;
   1:L PR[91] R[100]mm/sec CNT100;
   1:  PR[GP1:91,1] = PR[GP1:90,1] + -13.014;
   1:  PR[GP1:91,2] = PR[GP1:90,2] + 19.616;
   1:L PR[91] R[100]mm/sec CNT100;
   1:  PR[GP1:91,1] = PR[GP1:90,1] + -15.605;
   1:  PR[GP1:91,2] = PR[GP1:90,2] + 19.969;
   1:L PR[91] R[100]mm/sec CNT100;
   1:  PR[GP1:91,1] = PR[GP1:90,1] + -17.689;
   1:  PR[GP1:91,2] = PR[GP1:90,2] + 19.859;
   1:L PR[91] R[100]mm/sec CNT100;
   1:  PR[GP1:91,1] = PR[GP1:90,1] + -19.849;
   1:  PR[GP1:91,2] = PR[GP1:90,2] + 19.604;
   1:L PR[91] R[100]mm/sec CNT100;
   1:  PR[GP1:91,1] = PR[GP1:90,1] + -22.022;
   1:  PR[GP1:91,2] = PR[GP1:90,2] + 19.153;
   1:L PR[91] R[100]mm/sec CNT100;
   1:  PR[GP1:91,1] = PR[GP1:90,1] + -24.414;
   1:  PR[GP1:91,2] = PR[GP1:90,2] + 18.265;
   1:L PR[91] R[100]mm/sec CNT100;
   1:  PR[GP1:91,1] = PR[GP1:90,1] + -25.877;
   1:  PR[GP1:91,2] = PR[GP1:90,2] + 17.693;
   1:L PR[91] R[100]mm/sec CNT100;
   1:  PR[GP1:91,1] = PR[GP1:90,1] + -28.113;
   1:  PR[GP1:91,2] = PR[GP1:90,2] + 16.441;
   1:L PR[91] R[100]mm/sec CNT100;
   1:  PR[GP1:91,1] = PR[GP1:90,1] + -30.422;
   1:  PR[GP1:91,2] = PR[GP1:90,2] + 14.644;
   1:L PR[91] R[100]mm/sec CNT100;
   1:  PR[GP1:91,1] = PR[GP1:90,1] + -31.215;
   1:  PR[GP1:91,2] = PR[GP1:90,2] + 14.066;
   1:L PR[91] R[100]mm/sec CNT100;
   1:  PR[GP1:91,1] = PR[GP1:90,1] + -33.133;
   1:  PR[GP1:91,2] = PR[GP1:90,2] + 11.994;
   1:L PR[91] R[100]mm/sec CNT100;
   1:  PR[GP1:91,1] = PR[GP1:90,1] + -33.564;
   1:  PR[GP1:91,2] = PR[GP1:90,2] + 11.460;
   1:L PR[91] R[100]mm/sec CNT100;
   1:  PR[GP1:91,1] = PR[GP1:90,1] + -35.171;
   1:  PR[GP1:91,2] = PR[GP1:90,2] + 9.018;
   1:L PR[91] R[100]mm/sec CNT100;
   1:  PR[GP1:91,1] = PR[GP1:90,1] + -36.621;
   1:  PR[GP1:91,2] = PR[GP1:90,2] + 5.773;
   1:L PR[91] R[100]mm/sec CNT100;
   1:  PR[GP1:91,1] = PR[GP1:90,1] + -37.347;
   1:  PR[GP1:91,2] = PR[GP1:90,2] + 2.970;
   1:L PR[91] R[100]mm/sec CNT100;
   1:  PR[GP1:91,1] = PR[GP1:90,1] + -37.596;
   1:  PR[GP1:91,2] = PR[GP1:90,2] + -0.139;
   1:L PR[91] R[100]mm/sec CNT100;
   1:  PR[GP1:91,1] = PR[GP1:90,1] + -37.625;
   1:  PR[GP1:91,2] = PR[GP1:90,2] + -0.354;
   1:L PR[91] R[100]mm/sec CNT100;
   1:  PR[GP1:91,1] = PR[GP1:90,1] + -37.389;
   1:  PR[GP1:91,2] = PR[GP1:90,2] + -3.326;
   1:L PR[91] R[100]mm/sec CNT100;
   1:  PR[GP1:91,1] = PR[GP1:90,1] + -37.357;
   1:  PR[GP1:91,2] = PR[GP1:90,2] + -3.553;
   1:L PR[91] R[100]mm/sec CNT100;
   1:  PR[GP1:91,1] = PR[GP1:90,1] + -36.621;
   1:  PR[GP1:91,2] = PR[GP1:90,2] + -6.397;
   1:L PR[91] R[100]mm/sec CNT100;
   1:  PR[GP1:91,1] = PR[GP1:90,1] + -35.354;
   1:  PR[GP1:91,2] = PR[GP1:90,2] + -9.220;
   1:L PR[91] R[100]mm/sec CNT100;
   1:  PR[GP1:91,1] = PR[GP1:90,1] + -35.167;
   1:  PR[GP1:91,2] = PR[GP1:90,2] + -9.647;
   1:L PR[91] R[100]mm/sec CNT100;
   1:  PR[GP1:91,1] = PR[GP1:90,1] + -33.563;
   1:  PR[GP1:91,2] = PR[GP1:90,2] + -12.085;
   1:L PR[91] R[100]mm/sec CNT100;
   1:  PR[GP1:91,1] = PR[GP1:90,1] + -33.132;
   1:  PR[GP1:91,2] = PR[GP1:90,2] + -12.620;
   1:L PR[91] R[100]mm/sec CNT100;
   1:  PR[GP1:91,1] = PR[GP1:90,1] + -31.195;
   1:  PR[GP1:91,2] = PR[GP1:90,2] + -14.711;
   1:L PR[91] R[100]mm/sec CNT100;
   1:  PR[GP1:91,1] = PR[GP1:90,1] + -29.091;
   1:  PR[GP1:91,2] = PR[GP1:90,2] + -16.358;
   1:L PR[91] R[100]mm/sec CNT100;
   1:  PR[GP1:91,1] = PR[GP1:90,1] + -28.128;
   1:  PR[GP1:91,2] = PR[GP1:90,2] + -17.056;
   1:L PR[91] R[100]mm/sec CNT100;
   1:  PR[GP1:91,1] = PR[GP1:90,1] + -25.882;
   1:  PR[GP1:91,2] = PR[GP1:90,2] + -18.314;
   1:L PR[91] R[100]mm/sec CNT100;
   1:  PR[GP1:91,1] = PR[GP1:90,1] + -23.637;
   1:  PR[GP1:91,2] = PR[GP1:90,2] + -19.144;
   1:L PR[91] R[100]mm/sec CNT100;
   1:  PR[GP1:91,1] = PR[GP1:90,1] + -21.998;
   1:  PR[GP1:91,2] = PR[GP1:90,2] + -19.783;
   1:L PR[91] R[100]mm/sec CNT100;
   1:  PR[GP1:91,1] = PR[GP1:90,1] + -19.837;
   1:  PR[GP1:91,2] = PR[GP1:90,2] + -20.231;
   1:L PR[91] R[100]mm/sec CNT100;
   1:  PR[GP1:91,1] = PR[GP1:90,1] + -17.672;
   1:  PR[GP1:91,2] = PR[GP1:90,2] + -20.483;
   1:L PR[91] R[100]mm/sec CNT100;
   1:  PR[GP1:91,1] = PR[GP1:90,1] + -15.560;
   1:  PR[GP1:91,2] = PR[GP1:90,2] + -20.595;
   1:L PR[91] R[100]mm/sec CNT100;
   1:  PR[GP1:91,1] = PR[GP1:90,1] + -13.684;
   1:  PR[GP1:91,2] = PR[GP1:90,2] + -20.406;
   1:L PR[91] R[100]mm/sec CNT100;
   1:  PR[GP1:91,1] = PR[GP1:90,1] + -10.990;
   1:  PR[GP1:91,2] = PR[GP1:90,2] + -20.029;
   1:L PR[91] R[100]mm/sec CNT100;
   1:  PR[GP1:91,1] = PR[GP1:90,1] + -9.354;
   1:  PR[GP1:91,2] = PR[GP1:90,2] + -19.606;
   1:L PR[91] R[100]mm/sec CNT100;
   1:  PR[GP1:91,1] = PR[GP1:90,1] + -7.890;
   1:  PR[GP1:91,2] = PR[GP1:90,2] + -18.964;
   1:L PR[91] R[100]mm/sec CNT100;
   1:  PR[GP1:91,1] = PR[GP1:90,1] + -4.902;
   1:  PR[GP1:91,2] = PR[GP1:90,2] + -17.690;
   1:L PR[91] R[100]mm/sec CNT100;
   1:  PR[GP1:91,1] = PR[GP1:90,1] + -3.757;
   1:  PR[GP1:91,2] = PR[GP1:90,2] + -16.958;
   1:L PR[91] R[100]mm/sec CNT100;
   1:  PR[GP1:91,1] = PR[GP1:90,1] + -2.887;
   1:  PR[GP1:91,2] = PR[GP1:90,2] + -16.331;
   1:L PR[91] R[100]mm/sec CNT100;
   1:  PR[GP1:91,1] = PR[GP1:90,1] + -1.703;
   1:  PR[GP1:91,2] = PR[GP1:90,2] + -15.294;
   1:L PR[91] R[100]mm/sec CNT100;
   1:  PR[GP1:91,1] = PR[GP1:90,1] + -1.035;
   1:  PR[GP1:91,2] = PR[GP1:90,2] + -15.066;
   1:L PR[91] R[100]mm/sec CNT100;
   1:  PR[GP1:91,1] = PR[GP1:90,1] + -0.337;
   1:  PR[GP1:91,2] = PR[GP1:90,2] + -14.534;
   1:L PR[91] R[100]mm/sec CNT100;
   1:  PR[GP1:91,1] = PR[GP1:90,1] + 0.674;
   1:  PR[GP1:91,2] = PR[GP1:90,2] + -14.893;
   1:L PR[91] R[100]mm/sec CNT100;
   1:  PR[GP1:91,1] = PR[GP1:90,1] + 1.612;
   1:  PR[GP1:91,2] = PR[GP1:90,2] + -15.061;
   1:L PR[91] R[100]mm/sec CNT100;
   1:  PR[GP1:91,1] = PR[GP1:90,1] + 1.833;
   1:  PR[GP1:91,2] = PR[GP1:90,2] + -15.312;
   1:L PR[91] R[100]mm/sec CNT100;
   1:  PR[GP1:91,1] = PR[GP1:90,1] + 1.979;
   1:  PR[GP1:91,2] = PR[GP1:90,2] + -15.400;
   1:L PR[91] R[100]mm/sec CNT100;
   1:  PR[GP1:91,1] = PR[GP1:90,1] + 3.016;
   1:  PR[GP1:91,2] = PR[GP1:90,2] + -16.310;
   1:L PR[91] R[100]mm/sec CNT100;
   1:  PR[GP1:91,1] = PR[GP1:90,1] + 3.637;
   1:  PR[GP1:91,2] = PR[GP1:90,2] + -16.707;
   1:L PR[91] R[100]mm/sec CNT100;
   1:  PR[GP1:91,1] = PR[GP1:90,1] + 4.227;
   1:  PR[GP1:91,2] = PR[GP1:90,2] + -17.128;
   1:L PR[91] R[100]mm/sec CNT100;
   1:  PR[GP1:91,1] = PR[GP1:90,1] + 5.073;
   1:  PR[GP1:91,2] = PR[GP1:90,2] + -17.699;
   1:L PR[91] R[100]mm/sec CNT100;
   1:  PR[GP1:91,1] = PR[GP1:90,1] + 9.499;
   1:  PR[GP1:91,2] = PR[GP1:90,2] + -19.600;
   1:L PR[91] R[100]mm/sec CNT100;
   1:  PR[GP1:91,1] = PR[GP1:90,1] + 11.120;
   1:  PR[GP1:91,2] = PR[GP1:90,2] + -20.021;
   1:L PR[91] R[100]mm/sec CNT100;
   1:  PR[GP1:91,1] = PR[GP1:90,1] + 13.140;
   1:  PR[GP1:91,2] = PR[GP1:90,2] + -20.232;
   1:L PR[91] R[100]mm/sec CNT100;
   1:  PR[GP1:91,1] = PR[GP1:90,1] + 15.737;
   1:  PR[GP1:91,2] = PR[GP1:90,2] + -20.593;
   1:L PR[91] R[100]mm/sec CNT100;
   1:  PR[GP1:91,1] = PR[GP1:90,1] + 17.811;
   1:  PR[GP1:91,2] = PR[GP1:90,2] + -20.486;
   1:L PR[91] R[100]mm/sec CNT100;
   1:  PR[GP1:91,1] = PR[GP1:90,1] + 19.977;
   1:  PR[GP1:91,2] = PR[GP1:90,2] + -20.233;
   1:L PR[91] R[100]mm/sec CNT100;
   1:  PR[GP1:91,1] = PR[GP1:90,1] + 22.147;
   1:  PR[GP1:91,2] = PR[GP1:90,2] + -19.784;
   1:L PR[91] R[100]mm/sec CNT100;
   1:  PR[GP1:91,1] = PR[GP1:90,1] + 24.544;
   1:  PR[GP1:91,2] = PR[GP1:90,2] + -18.899;
   1:L PR[91] R[100]mm/sec CNT100;
   1:  PR[GP1:91,1] = PR[GP1:90,1] + 26.014;
   1:  PR[GP1:91,2] = PR[GP1:90,2] + -18.327;
   1:L PR[91] R[100]mm/sec CNT100;
   1:  PR[GP1:91,1] = PR[GP1:90,1] + 28.239;
   1:  PR[GP1:91,2] = PR[GP1:90,2] + -17.087;
   1:L PR[91] R[100]mm/sec CNT100;
   1:  PR[GP1:91,1] = PR[GP1:90,1] + 30.530;
   1:  PR[GP1:91,2] = PR[GP1:90,2] + -15.312;
   1:L PR[91] R[100]mm/sec CNT100;
   1:  PR[GP1:91,1] = PR[GP1:90,1] + 31.328;
   1:  PR[GP1:91,2] = PR[GP1:90,2] + -14.732;
   1:L PR[91] R[100]mm/sec CNT100;
   1:  PR[GP1:91,1] = PR[GP1:90,1] + 33.251;
   1:  PR[GP1:91,2] = PR[GP1:90,2] + -12.658;
   1:L PR[91] R[100]mm/sec CNT100;
   1:  PR[GP1:91,1] = PR[GP1:90,1] + 33.686;
   1:  PR[GP1:91,2] = PR[GP1:90,2] + -12.118;
   1:L PR[91] R[100]mm/sec CNT100;
   1:  PR[GP1:91,1] = PR[GP1:90,1] + 35.315;
   1:  PR[GP1:91,2] = PR[GP1:90,2] + -9.656;
   1:L PR[91] R[100]mm/sec CNT100;
   1:  PR[GP1:91,1] = PR[GP1:90,1] + 36.629;
   1:  PR[GP1:91,2] = PR[GP1:90,2] + -6.763;
   1:L PR[91] R[100]mm/sec CNT100;
   1:  PR[GP1:91,1] = PR[GP1:90,1] + 36.761;
   1:  PR[GP1:91,2] = PR[GP1:90,2] + -6.463;
   1:L PR[91] R[100]mm/sec CNT100;
   1:  PR[GP1:91,1] = PR[GP1:90,1] + 37.490;
   1:  PR[GP1:91,2] = PR[GP1:90,2] + -3.687;
   1:L PR[91] R[100]mm/sec CNT100;
   1:  PR[GP1:91,1] = PR[GP1:90,1] + 37.753;
   1:  PR[GP1:91,2] = PR[GP1:90,2] + -0.485;
   1:L PR[91] R[100]mm/sec CNT100;
   1:  PR[GP1:91,1] = PR[GP1:90,1] + 37.782;
   1:  PR[GP1:91,2] = PR[GP1:90,2] + -0.271;
   1:L PR[91] R[100]mm/sec CNT100;
   1:  PR[GP1:91,1] = PR[GP1:90,1] + 37.532;
   1:  PR[GP1:91,2] = PR[GP1:90,2] + 2.795;
   1:L PR[91] R[100]mm/sec CNT100;
   1:  PR[GP1:91,1] = PR[GP1:90,1] + 37.500;
   1:  PR[GP1:91,2] = PR[GP1:90,2] + 3.023;
   1:L PR[91] R[100]mm/sec CNT100;
   1:  PR[GP1:91,1] = PR[GP1:90,1] + 36.763;
   1:  PR[GP1:91,2] = PR[GP1:90,2] + 5.831;
   1:L PR[91] R[100]mm/sec CNT100;
   1:  PR[GP1:91,1] = PR[GP1:90,1] + 35.316;
   1:  PR[GP1:91,2] = PR[GP1:90,2] + 9.032;
   1:L PR[91] R[100]mm/sec CNT100;
   1:  PR[GP1:91,1] = PR[GP1:90,1] + 33.687;
   1:  PR[GP1:91,2] = PR[GP1:90,2] + 11.493;
   1:L PR[91] R[100]mm/sec CNT100;
   1:  PR[GP1:91,1] = PR[GP1:90,1] + 33.253;
   1:  PR[GP1:91,2] = PR[GP1:90,2] + 12.032;
   1:L PR[91] R[100]mm/sec CNT100;
   1:  PR[GP1:91,1] = PR[GP1:90,1] + 31.314;
   1:  PR[GP1:91,2] = PR[GP1:90,2] + 14.124;
   1:L PR[91] R[100]mm/sec CNT100;
   1:  PR[GP1:91,1] = PR[GP1:90,1] + 29.228;
   1:  PR[GP1:91,2] = PR[GP1:90,2] + 15.750;
   1:L PR[91] R[100]mm/sec CNT100;
   1:  PR[GP1:91,1] = PR[GP1:90,1] + 28.265;
   1:  PR[GP1:91,2] = PR[GP1:90,2] + 16.449;
   1:L PR[91] R[100]mm/sec CNT100;
   1:  PR[GP1:91,1] = PR[GP1:90,1] + 26.032;
   1:  PR[GP1:91,2] = PR[GP1:90,2] + 17.693;
   1:L PR[91] R[100]mm/sec CNT100;
   1:  PR[GP1:91,1] = PR[GP1:90,1] + 23.783;
   1:  PR[GP1:91,2] = PR[GP1:90,2] + 18.520;
   1:L PR[91] R[100]mm/sec CNT100;
   1:  PR[GP1:91,1] = PR[GP1:90,1] + 22.146;
   1:  PR[GP1:91,2] = PR[GP1:90,2] + 19.160;
   1:L PR[91] R[100]mm/sec CNT100;
   1:  PR[GP1:91,1] = PR[GP1:90,1] + 19.988;
   1:  PR[GP1:91,2] = PR[GP1:90,2] + 19.606;
   1:L PR[91] R[100]mm/sec CNT100;
   1:  PR[GP1:91,1] = PR[GP1:90,1] + 17.828;
   1:  PR[GP1:91,2] = PR[GP1:90,2] + 19.862;
   1:L PR[91] R[100]mm/sec CNT100;
   1:  PR[GP1:91,1] = PR[GP1:90,1] + 15.729;
   1:  PR[GP1:91,2] = PR[GP1:90,2] + 19.971;
   1:L PR[91] R[100]mm/sec CNT100;
   1:  PR[GP1:91,1] = PR[GP1:90,1] + 13.857;
   1:  PR[GP1:91,2] = PR[GP1:90,2] + 19.781;
   1:L PR[91] R[100]mm/sec CNT100;
   1:  PR[GP1:91,1] = PR[GP1:90,1] + 11.168;
   1:  PR[GP1:91,2] = PR[GP1:90,2] + 19.409;
   1:L PR[91] R[100]mm/sec CNT100;
   1:  PR[GP1:91,1] = PR[GP1:90,1] + 9.530;
   1:  PR[GP1:91,2] = PR[GP1:90,2] + 18.985;
   1:L PR[91] R[100]mm/sec CNT100;
   1:  PR[GP1:91,1] = PR[GP1:90,1] + 8.064;
   1:  PR[GP1:91,2] = PR[GP1:90,2] + 18.343;
   1:L PR[91] R[100]mm/sec CNT100;
   1:  PR[GP1:91,1] = PR[GP1:90,1] + 5.139;
   1:  PR[GP1:91,2] = PR[GP1:90,2] + 17.121;
   1:L PR[91] R[100]mm/sec CNT100;
   1:  PR[GP1:91,1] = PR[GP1:90,1] + 3.965;
   1:  PR[GP1:91,2] = PR[GP1:90,2] + 16.371;
   1:L PR[91] R[100]mm/sec CNT100;
   1:  PR[GP1:91,1] = PR[GP1:90,1] + 3.405;
   1:  PR[GP1:91,2] = PR[GP1:90,2] + 15.985;
   1:L PR[91] R[100]mm/sec CNT100;
   1:  PR[GP1:91,1] = PR[GP1:90,1] + 2.387;
   1:  PR[GP1:91,2] = PR[GP1:90,2] + 15.179;
   1:L PR[91] R[100]mm/sec CNT100;
   1:  PR[GP1:91,1] = PR[GP1:90,1] + 2.008;
   1:  PR[GP1:91,2] = PR[GP1:90,2] + 14.843;
   1:L PR[91] R[100]mm/sec CNT100;
   1:  PR[GP1:91,1] = PR[GP1:90,1] + 1.924;
   1:  PR[GP1:91,2] = PR[GP1:90,2] + 14.787;
   1:L PR[91] R[100]mm/sec CNT100;
   1:  PR[GP1:91,1] = PR[GP1:90,1] + 1.541;
   1:  PR[GP1:91,2] = PR[GP1:90,2] + 14.416;
   1:L PR[91] R[100]mm/sec CNT100;
   1:  PR[GP1:91,1] = PR[GP1:90,1] + 0.779;
   1:  PR[GP1:91,2] = PR[GP1:90,2] + 14.285;
   1:L PR[91] R[100]mm/sec CNT100;
   1:  PR[GP1:91,1] = PR[GP1:90,1] + 0.419;
   1:  PR[GP1:91,2] = PR[GP1:90,2] + 14.088;
   1:L PR[91] R[100]mm/sec CNT100;
   1:  PR[GP1:91,1] = PR[GP1:90,1] + -0.391;
   1:L PR[91] R[100]mm/sec CNT100;
   1:  PR[91] = PR[90];
   1:  PR[GP1:91,1] = PR[GP1:90,1] + -1.750;
   1:  PR[GP1:91,2] = PR[GP1:90,2] + 15.019;
   1:  PR[GP1:91,3] = PR[GP1:90,3] + 33.245;
   1:L PR[91] R[100]mm/sec CNT100;
   1:  PR[GP1:91,1] = PR[GP1:90,1] + -1.966;
   1:  PR[GP1:91,2] = PR[GP1:90,2] + 15.226;
   1:L PR[91] R[100]mm/sec CNT100;
   1:  PR[GP1:91,1] = PR[GP1:90,1] + -3.004;
   1:  PR[GP1:91,2] = PR[GP1:90,2] + 16.046;
   1:L PR[91] R[100]mm/sec CNT100;
   1:  PR[GP1:91,1] = PR[GP1:90,1] + -3.762;
   1:  PR[GP1:91,2] = PR[GP1:90,2] + 16.531;
   1:L PR[91] R[100]mm/sec CNT100;
   1:  PR[GP1:91,1] = PR[GP1:90,1] + -4.723;
   1:  PR[GP1:91,2] = PR[GP1:90,2] + 17.176;
   1:L PR[91] R[100]mm/sec CNT100;
   1:  PR[GP1:91,1] = PR[GP1:90,1] + -6.056;
   1:  PR[GP1:91,2] = PR[GP1:90,2] + 17.758;
   1:L PR[91] R[100]mm/sec CNT100;
   1:  PR[GP1:91,1] = PR[GP1:90,1] + -9.172;
   1:  PR[GP1:91,2] = PR[GP1:90,2] + 19.064;
   1:L PR[91] R[100]mm/sec CNT100;
   1:  PR[GP1:91,1] = PR[GP1:90,1] + -10.666;
   1:  PR[GP1:91,2] = PR[GP1:90,2] + 19.451;
   1:L PR[91] R[100]mm/sec CNT100;
   1:  PR[GP1:91,1] = PR[GP1:90,1] + -12.540;
   1:  PR[GP1:91,2] = PR[GP1:90,2] + 19.646;
   1:L PR[91] R[100]mm/sec CNT100;
   1:  PR[GP1:91,1] = PR[GP1:90,1] + -15.381;
   1:  PR[GP1:91,2] = PR[GP1:90,2] + 20.034;
   1:L PR[91] R[100]mm/sec CNT100;
   1:  PR[GP1:91,1] = PR[GP1:90,1] + -17.322;
   1:  PR[GP1:91,2] = PR[GP1:90,2] + 19.931;
   1:L PR[91] R[100]mm/sec CNT100;
   1:  PR[GP1:91,1] = PR[GP1:90,1] + -19.724;
   1:  PR[GP1:91,2] = PR[GP1:90,2] + 19.647;
   1:L PR[91] R[100]mm/sec CNT100;
   1:  PR[GP1:91,1] = PR[GP1:90,1] + -21.764;
   1:  PR[GP1:91,2] = PR[GP1:90,2] + 19.224;
   1:L PR[91] R[100]mm/sec CNT100;
   1:  PR[GP1:91,1] = PR[GP1:90,1] + -24.013;
   1:  PR[GP1:91,2] = PR[GP1:90,2] + 18.389;
   1:L PR[91] R[100]mm/sec CNT100;
   1:  PR[GP1:91,1] = PR[GP1:90,1] + -25.716;
   1:  PR[GP1:91,2] = PR[GP1:90,2] + 17.723;
   1:L PR[91] R[100]mm/sec CNT100;
   1:  PR[GP1:91,1] = PR[GP1:90,1] + -27.825;
   1:  PR[GP1:91,2] = PR[GP1:90,2] + 16.541;
   1:L PR[91] R[100]mm/sec CNT100;
   1:  PR[GP1:91,1] = PR[GP1:90,1] + -30.010;
   1:  PR[GP1:91,2] = PR[GP1:90,2] + 14.841;
   1:L PR[91] R[100]mm/sec CNT100;
   1:  PR[GP1:91,1] = PR[GP1:90,1] + -31.019;
   1:  PR[GP1:91,2] = PR[GP1:90,2] + 14.106;
   1:L PR[91] R[100]mm/sec CNT100;
   1:  PR[GP1:91,1] = PR[GP1:90,1] + -32.838;
   1:  PR[GP1:91,2] = PR[GP1:90,2] + 12.142;
   1:L PR[91] R[100]mm/sec CNT100;
   1:  PR[GP1:91,1] = PR[GP1:90,1] + -33.428;
   1:  PR[GP1:91,2] = PR[GP1:90,2] + 11.409;
   1:L PR[91] R[100]mm/sec CNT100;
   1:  PR[GP1:91,1] = PR[GP1:90,1] + -34.956;
   1:  PR[GP1:91,2] = PR[GP1:90,2] + 9.087;
   1:L PR[91] R[100]mm/sec CNT100;
   1:  PR[GP1:91,1] = PR[GP1:90,1] + -36.446;
   1:  PR[GP1:91,2] = PR[GP1:90,2] + 5.748;
   1:L PR[91] R[100]mm/sec CNT100;
   1:  PR[GP1:91,1] = PR[GP1:90,1] + -37.137;
   1:  PR[GP1:91,2] = PR[GP1:90,2] + 3.081;
   1:L PR[91] R[100]mm/sec CNT100;
   1:  PR[GP1:91,1] = PR[GP1:90,1] + -37.374;
   1:  PR[GP1:91,2] = PR[GP1:90,2] + 0.115;
   1:L PR[91] R[100]mm/sec CNT100;
   1:  PR[GP1:91,1] = PR[GP1:90,1] + -37.439;
   1:  PR[GP1:91,2] = PR[GP1:90,2] + -0.354;
   1:L PR[91] R[100]mm/sec CNT100;
   1:  PR[GP1:91,1] = PR[GP1:90,1] + -37.214;
   1:  PR[GP1:91,2] = PR[GP1:90,2] + -3.186;
   1:L PR[91] R[100]mm/sec CNT100;
   1:  PR[GP1:91,1] = PR[GP1:90,1] + -37.147;
   1:  PR[GP1:91,2] = PR[GP1:90,2] + -3.665;
   1:L PR[91] R[100]mm/sec CNT100;
   1:  PR[GP1:91,1] = PR[GP1:90,1] + -36.446;
   1:  PR[GP1:91,2] = PR[GP1:90,2] + -6.371;
   1:L PR[91] R[100]mm/sec CNT100;
   1:  PR[GP1:91,1] = PR[GP1:90,1] + -35.239;
   1:  PR[GP1:91,2] = PR[GP1:90,2] + -9.063;
   1:L PR[91] R[100]mm/sec CNT100;
   1:  PR[GP1:91,1] = PR[GP1:90,1] + -34.952;
   1:  PR[GP1:91,2] = PR[GP1:90,2] + -9.717;
   1:L PR[91] R[100]mm/sec CNT100;
   1:  PR[GP1:91,1] = PR[GP1:90,1] + -33.427;
   1:  PR[GP1:91,2] = PR[GP1:90,2] + -12.034;
   1:L PR[91] R[100]mm/sec CNT100;
   1:  PR[GP1:91,1] = PR[GP1:90,1] + -32.835;
   1:  PR[GP1:91,2] = PR[GP1:90,2] + -12.768;
   1:L PR[91] R[100]mm/sec CNT100;
   1:  PR[GP1:91,1] = PR[GP1:90,1] + -30.998;
   1:  PR[GP1:91,2] = PR[GP1:90,2] + -14.752;
   1:L PR[91] R[100]mm/sec CNT100;
   1:  PR[GP1:91,1] = PR[GP1:90,1] + -29.002;
   1:  PR[GP1:91,2] = PR[GP1:90,2] + -16.314;
   1:L PR[91] R[100]mm/sec CNT100;
   1:  PR[GP1:91,1] = PR[GP1:90,1] + -27.839;
   1:  PR[GP1:91,2] = PR[GP1:90,2] + -17.157;
   1:L PR[91] R[100]mm/sec CNT100;
   1:  PR[GP1:91,1] = PR[GP1:90,1] + -25.720;
   1:  PR[GP1:91,2] = PR[GP1:90,2] + -18.345;
   1:L PR[91] R[100]mm/sec CNT100;
   1:  PR[GP1:91,1] = PR[GP1:90,1] + -23.597;
   1:  PR[GP1:91,2] = PR[GP1:90,2] + -19.129;
   1:L PR[91] R[100]mm/sec CNT100;
   1:  PR[GP1:91,1] = PR[GP1:90,1] + -21.738;
   1:  PR[GP1:91,2] = PR[GP1:90,2] + -19.854;
   1:L PR[91] R[100]mm/sec CNT100;
   1:  PR[GP1:91,1] = PR[GP1:90,1] + -19.710;
   1:  PR[GP1:91,2] = PR[GP1:90,2] + -20.274;
   1:L PR[91] R[100]mm/sec CNT100;
   1:  PR[GP1:91,1] = PR[GP1:90,1] + -17.303;
   1:  PR[GP1:91,2] = PR[GP1:90,2] + -20.555;
   1:L PR[91] R[100]mm/sec CNT100;
   1:  PR[GP1:91,1] = PR[GP1:90,1] + -15.334;
   1:  PR[GP1:91,2] = PR[GP1:90,2] + -20.659;
   1:L PR[91] R[100]mm/sec CNT100;
   1:  PR[GP1:91,1] = PR[GP1:90,1] + -13.585;
   1:  PR[GP1:91,2] = PR[GP1:90,2] + -20.483;
   1:L PR[91] R[100]mm/sec CNT100;
   1:  PR[GP1:91,1] = PR[GP1:90,1] + -10.663;
   1:  PR[GP1:91,2] = PR[GP1:90,2] + -20.074;
   1:L PR[91] R[100]mm/sec CNT100;
   1:  PR[GP1:91,1] = PR[GP1:90,1] + -9.156;
   1:  PR[GP1:91,2] = PR[GP1:90,2] + -19.684;
   1:L PR[91] R[100]mm/sec CNT100;
   1:  PR[GP1:91,1] = PR[GP1:90,1] + -7.803;
   1:  PR[GP1:91,2] = PR[GP1:90,2] + -19.090;
   1:L PR[91] R[100]mm/sec CNT100;
   1:  PR[GP1:91,1] = PR[GP1:90,1] + -4.609;
   1:  PR[GP1:91,2] = PR[GP1:90,2] + -17.729;
   1:L PR[91] R[100]mm/sec CNT100;
   1:  PR[GP1:91,1] = PR[GP1:90,1] + -3.572;
   1:  PR[GP1:91,2] = PR[GP1:90,2] + -17.067;
   1:L PR[91] R[100]mm/sec CNT100;
   1:  PR[GP1:91,1] = PR[GP1:90,1] + -2.643;
   1:  PR[GP1:91,2] = PR[GP1:90,2] + -16.396;
   1:L PR[91] R[100]mm/sec CNT100;
   1:  PR[GP1:91,1] = PR[GP1:90,1] + -1.685;
   1:  PR[GP1:91,2] = PR[GP1:90,2] + -15.558;
   1:L PR[91] R[100]mm/sec CNT100;
   1:  PR[GP1:91,1] = PR[GP1:90,1] + -0.884;
   1:  PR[GP1:91,2] = PR[GP1:90,2] + -15.285;
   1:L PR[91] R[100]mm/sec CNT100;
   1:  PR[GP1:91,1] = PR[GP1:90,1] + -0.313;
   1:  PR[GP1:91,2] = PR[GP1:90,2] + -14.848;
   1:L PR[91] R[100]mm/sec CNT100;
   1:  PR[GP1:91,1] = PR[GP1:90,1] + 0.513;
   1:  PR[GP1:91,2] = PR[GP1:90,2] + -15.142;
   1:L PR[91] R[100]mm/sec CNT100;
   1:  PR[GP1:91,1] = PR[GP1:90,1] + 1.632;
   1:  PR[GP1:91,2] = PR[GP1:90,2] + -15.342;
   1:L PR[91] R[100]mm/sec CNT100;
   1:  PR[GP1:91,1] = PR[GP1:90,1] + 1.864;
   1:  PR[GP1:91,2] = PR[GP1:90,2] + -15.606;
   1:L PR[91] R[100]mm/sec CNT100;
   1:  PR[GP1:91,1] = PR[GP1:90,1] + 1.960;
   1:  PR[GP1:91,2] = PR[GP1:90,2] + -15.664;
   1:L PR[91] R[100]mm/sec CNT100;
   1:  PR[GP1:91,1] = PR[GP1:90,1] + 2.771;
   1:  PR[GP1:91,2] = PR[GP1:90,2] + -16.374;
   1:L PR[91] R[100]mm/sec CNT100;
   1:  PR[GP1:91,1] = PR[GP1:90,1] + 3.240;
   1:  PR[GP1:91,2] = PR[GP1:90,2] + -16.675;
   1:L PR[91] R[100]mm/sec CNT100;
   1:  PR[GP1:91,1] = PR[GP1:90,1] + 3.869;
   1:  PR[GP1:91,2] = PR[GP1:90,2] + -17.123;
   1:L PR[91] R[100]mm/sec CNT100;
   1:  PR[GP1:91,1] = PR[GP1:90,1] + 4.780;
   1:  PR[GP1:91,2] = PR[GP1:90,2] + -17.738;
   1:L PR[91] R[100]mm/sec CNT100;
   1:  PR[GP1:91,1] = PR[GP1:90,1] + 9.302;
   1:  PR[GP1:91,2] = PR[GP1:90,2] + -19.679;
   1:L PR[91] R[100]mm/sec CNT100;
   1:  PR[GP1:91,1] = PR[GP1:90,1] + 10.793;
   1:  PR[GP1:91,2] = PR[GP1:90,2] + -20.065;
   1:L PR[91] R[100]mm/sec CNT100;
   1:  PR[GP1:91,1] = PR[GP1:90,1] + 12.664;
   1:  PR[GP1:91,2] = PR[GP1:90,2] + -20.262;
   1:L PR[91] R[100]mm/sec CNT100;
   1:  PR[GP1:91,1] = PR[GP1:90,1] + 15.511;
   1:  PR[GP1:91,2] = PR[GP1:90,2] + -20.658;
   1:L PR[91] R[100]mm/sec CNT100;
   1:  PR[GP1:91,1] = PR[GP1:90,1] + 17.443;
   1:  PR[GP1:91,2] = PR[GP1:90,2] + -20.557;
   1:L PR[91] R[100]mm/sec CNT100;
   1:  PR[GP1:91,1] = PR[GP1:90,1] + 19.851;
   1:  PR[GP1:91,2] = PR[GP1:90,2] + -20.277;
   1:L PR[91] R[100]mm/sec CNT100;
   1:  PR[GP1:91,1] = PR[GP1:90,1] + 21.888;
   1:  PR[GP1:91,2] = PR[GP1:90,2] + -19.855;
   1:L PR[91] R[100]mm/sec CNT100;
   1:  PR[GP1:91,1] = PR[GP1:90,1] + 24.142;
   1:  PR[GP1:91,2] = PR[GP1:90,2] + -19.022;
   1:L PR[91] R[100]mm/sec CNT100;
   1:  PR[GP1:91,1] = PR[GP1:90,1] + 25.852;
   1:  PR[GP1:91,2] = PR[GP1:90,2] + -18.358;
   1:L PR[91] R[100]mm/sec CNT100;
   1:  PR[GP1:91,1] = PR[GP1:90,1] + 27.952;
   1:  PR[GP1:91,2] = PR[GP1:90,2] + -17.187;
   1:L PR[91] R[100]mm/sec CNT100;
   1:  PR[GP1:91,1] = PR[GP1:90,1] + 30.119;
   1:  PR[GP1:91,2] = PR[GP1:90,2] + -15.508;
   1:L PR[91] R[100]mm/sec CNT100;
   1:  PR[GP1:91,1] = PR[GP1:90,1] + 31.133;
   1:  PR[GP1:91,2] = PR[GP1:90,2] + -14.771;
   1:L PR[91] R[100]mm/sec CNT100;
   1:  PR[GP1:91,1] = PR[GP1:90,1] + 32.956;
   1:  PR[GP1:91,2] = PR[GP1:90,2] + -12.805;
   1:L PR[91] R[100]mm/sec CNT100;
   1:  PR[GP1:91,1] = PR[GP1:90,1] + 33.551;
   1:  PR[GP1:91,2] = PR[GP1:90,2] + -12.066;
   1:L PR[91] R[100]mm/sec CNT100;
   1:  PR[GP1:91,1] = PR[GP1:90,1] + 35.101;
   1:  PR[GP1:91,2] = PR[GP1:90,2] + -9.725;
   1:L PR[91] R[100]mm/sec CNT100;
   1:  PR[GP1:91,1] = PR[GP1:90,1] + 36.351;
   1:  PR[GP1:91,2] = PR[GP1:90,2] + -6.972;
   1:L PR[91] R[100]mm/sec CNT100;
   1:  PR[GP1:91,1] = PR[GP1:90,1] + 36.587;
   1:  PR[GP1:91,2] = PR[GP1:90,2] + -6.435;
   1:L PR[91] R[100]mm/sec CNT100;
   1:  PR[GP1:91,1] = PR[GP1:90,1] + 37.280;
   1:  PR[GP1:91,2] = PR[GP1:90,2] + -3.795;
   1:L PR[91] R[100]mm/sec CNT100;
   1:  PR[GP1:91,1] = PR[GP1:90,1] + 37.531;
   1:  PR[GP1:91,2] = PR[GP1:90,2] + -0.740;
   1:L PR[91] R[100]mm/sec CNT100;
   1:  PR[GP1:91,1] = PR[GP1:90,1] + 37.596;
   1:  PR[GP1:91,2] = PR[GP1:90,2] + -0.271;
   1:L PR[91] R[100]mm/sec CNT100;
   1:  PR[GP1:91,1] = PR[GP1:90,1] + 37.358;
   1:  PR[GP1:91,2] = PR[GP1:90,2] + 2.651;
   1:L PR[91] R[100]mm/sec CNT100;
   1:  PR[GP1:91,1] = PR[GP1:90,1] + 37.291;
   1:  PR[GP1:91,2] = PR[GP1:90,2] + 3.131;
   1:L PR[91] R[100]mm/sec CNT100;
   1:  PR[GP1:91,1] = PR[GP1:90,1] + 36.589;
   1:  PR[GP1:91,2] = PR[GP1:90,2] + 5.804;
   1:L PR[91] R[100]mm/sec CNT100;
   1:  PR[GP1:91,1] = PR[GP1:90,1] + 35.101;
   1:  PR[GP1:91,2] = PR[GP1:90,2] + 9.100;
   1:L PR[91] R[100]mm/sec CNT100;
   1:  PR[GP1:91,1] = PR[GP1:90,1] + 33.552;
   1:  PR[GP1:91,2] = PR[GP1:90,2] + 11.440;
   1:L PR[91] R[100]mm/sec CNT100;
   1:  PR[GP1:91,1] = PR[GP1:90,1] + 32.959;
   1:  PR[GP1:91,2] = PR[GP1:90,2] + 12.178;
   1:L PR[91] R[100]mm/sec CNT100;
   1:  PR[GP1:91,1] = PR[GP1:90,1] + 31.120;
   1:  PR[GP1:91,2] = PR[GP1:90,2] + 14.162;
   1:L PR[91] R[100]mm/sec CNT100;
   1:  PR[GP1:91,1] = PR[GP1:90,1] + 29.140;
   1:  PR[GP1:91,2] = PR[GP1:90,2] + 15.704;
   1:L PR[91] R[100]mm/sec CNT100;
   1:  PR[GP1:91,1] = PR[GP1:90,1] + 27.979;
   1:  PR[GP1:91,2] = PR[GP1:90,2] + 16.549;
   1:L PR[91] R[100]mm/sec CNT100;
   1:  PR[GP1:91,1] = PR[GP1:90,1] + 25.871;
   1:  PR[GP1:91,2] = PR[GP1:90,2] + 17.723;
   1:L PR[91] R[100]mm/sec CNT100;
   1:  PR[GP1:91,1] = PR[GP1:90,1] + 23.744;
   1:  PR[GP1:91,2] = PR[GP1:90,2] + 18.504;
   1:L PR[91] R[100]mm/sec CNT100;
   1:  PR[GP1:91,1] = PR[GP1:90,1] + 21.888;
   1:  PR[GP1:91,2] = PR[GP1:90,2] + 19.230;
   1:L PR[91] R[100]mm/sec CNT100;
   1:  PR[GP1:91,1] = PR[GP1:90,1] + 19.864;
   1:  PR[GP1:91,2] = PR[GP1:90,2] + 19.649;
   1:L PR[91] R[100]mm/sec CNT100;
   1:  PR[GP1:91,1] = PR[GP1:90,1] + 17.462;
   1:  PR[GP1:91,2] = PR[GP1:90,2] + 19.933;
   1:L PR[91] R[100]mm/sec CNT100;
   1:  PR[GP1:91,1] = PR[GP1:90,1] + 15.505;
   1:  PR[GP1:91,2] = PR[GP1:90,2] + 20.035;
   1:L PR[91] R[100]mm/sec CNT100;
   1:  PR[GP1:91,1] = PR[GP1:90,1] + 13.759;
   1:  PR[GP1:91,2] = PR[GP1:90,2] + 19.858;
   1:L PR[91] R[100]mm/sec CNT100;
   1:  PR[GP1:91,1] = PR[GP1:90,1] + 10.843;
   1:  PR[GP1:91,2] = PR[GP1:90,2] + 19.455;
   1:L PR[91] R[100]mm/sec CNT100;
   1:  PR[GP1:91,1] = PR[GP1:90,1] + 9.334;
   1:  PR[GP1:91,2] = PR[GP1:90,2] + 19.064;
   1:L PR[91] R[100]mm/sec CNT100;
   1:  PR[GP1:91,1] = PR[GP1:90,1] + 7.979;
   1:  PR[GP1:91,2] = PR[GP1:90,2] + 18.471;
   1:L PR[91] R[100]mm/sec CNT100;
   1:  PR[GP1:91,1] = PR[GP1:90,1] + 4.851;
   1:  PR[GP1:91,2] = PR[GP1:90,2] + 17.164;
   1:L PR[91] R[100]mm/sec CNT100;
   1:  PR[GP1:91,1] = PR[GP1:90,1] + 3.782;
   1:  PR[GP1:91,2] = PR[GP1:90,2] + 16.481;
   1:L PR[91] R[100]mm/sec CNT100;
   1:  PR[GP1:91,1] = PR[GP1:90,1] + 3.184;
   1:  PR[GP1:91,2] = PR[GP1:90,2] + 16.068;
   1:L PR[91] R[100]mm/sec CNT100;
   1:  PR[GP1:91,1] = PR[GP1:90,1] + 2.112;
   1:  PR[GP1:91,2] = PR[GP1:90,2] + 15.220;
   1:L PR[91] R[100]mm/sec CNT100;
   1:  PR[GP1:91,1] = PR[GP1:90,1] + 1.543;
   1:  PR[GP1:91,2] = PR[GP1:90,2] + 14.693;
   1:L PR[91] R[100]mm/sec CNT100;
   1:  PR[GP1:91,1] = PR[GP1:90,1] + 0.620;
   1:  PR[GP1:91,2] = PR[GP1:90,2] + 14.535;
   1:L PR[91] R[100]mm/sec CNT100;
   1:  PR[GP1:91,1] = PR[GP1:90,1] + 0.378;
   1:  PR[GP1:91,2] = PR[GP1:90,2] + 14.403;
   1:L PR[91] R[100]mm/sec CNT100;
   1:  PR[GP1:91,1] = PR[GP1:90,1] + -0.366;
   1:L PR[91] R[100]mm/sec CNT100;
   1:  PR[91] = PR[90];
   1:  PR[GP1:91,1] = PR[GP1:90,1] + -1.654;
   1:  PR[GP1:91,2] = PR[GP1:90,2] + 15.236;
   1:  PR[GP1:91,3] = PR[GP1:90,3] + 33.855;
   1:L PR[91] R[100]mm/sec CNT100;
   1:  PR[GP1:91,1] = PR[GP1:90,1] + -2.784;
   1:  PR[GP1:91,2] = PR[GP1:90,2] + 16.130;
   1:L PR[91] R[100]mm/sec CNT100;
   1:  PR[GP1:91,1] = PR[GP1:90,1] + -3.408;
   1:  PR[GP1:91,2] = PR[GP1:90,2] + 16.530;
   1:L PR[91] R[100]mm/sec CNT100;
   1:  PR[GP1:91,1] = PR[GP1:90,1] + -4.436;
   1:  PR[GP1:91,2] = PR[GP1:90,2] + 17.219;
   1:L PR[91] R[100]mm/sec CNT100;
   1:  PR[GP1:91,1] = PR[GP1:90,1] + -5.640;
   1:  PR[GP1:91,2] = PR[GP1:90,2] + 17.745;
   1:L PR[91] R[100]mm/sec CNT100;
   1:  PR[GP1:91,1] = PR[GP1:90,1] + -8.977;
   1:  PR[GP1:91,2] = PR[GP1:90,2] + 19.143;
   1:L PR[91] R[100]mm/sec CNT100;
   1:  PR[GP1:91,1] = PR[GP1:90,1] + -10.341;
   1:  PR[GP1:91,2] = PR[GP1:90,2] + 19.496;
   1:L PR[91] R[100]mm/sec CNT100;
   1:  PR[GP1:91,1] = PR[GP1:90,1] + -12.067;
   1:  PR[GP1:91,2] = PR[GP1:90,2] + 19.676;
   1:L PR[91] R[100]mm/sec CNT100;
   1:  PR[GP1:91,1] = PR[GP1:90,1] + -15.157;
   1:  PR[GP1:91,2] = PR[GP1:90,2] + 20.098;
   1:L PR[91] R[100]mm/sec CNT100;
   1:  PR[GP1:91,1] = PR[GP1:90,1] + -16.955;
   1:  PR[GP1:91,2] = PR[GP1:90,2] + 20.003;
   1:L PR[91] R[100]mm/sec CNT100;
   1:  PR[GP1:91,1] = PR[GP1:90,1] + -19.599;
   1:  PR[GP1:91,2] = PR[GP1:90,2] + 19.690;
   1:L PR[91] R[100]mm/sec CNT100;
   1:  PR[GP1:91,1] = PR[GP1:90,1] + -21.505;
   1:  PR[GP1:91,2] = PR[GP1:90,2] + 19.294;
   1:L PR[91] R[100]mm/sec CNT100;
   1:  PR[GP1:91,1] = PR[GP1:90,1] + -23.612;
   1:  PR[GP1:91,2] = PR[GP1:90,2] + 18.513;
   1:L PR[91] R[100]mm/sec CNT100;
   1:  PR[GP1:91,1] = PR[GP1:90,1] + -25.554;
   1:  PR[GP1:91,2] = PR[GP1:90,2] + 17.753;
   1:L PR[91] R[100]mm/sec CNT100;
   1:  PR[GP1:91,1] = PR[GP1:90,1] + -27.537;
   1:  PR[GP1:91,2] = PR[GP1:90,2] + 16.642;
   1:L PR[91] R[100]mm/sec CNT100;
   1:  PR[GP1:91,1] = PR[GP1:90,1] + -29.598;
   1:  PR[GP1:91,2] = PR[GP1:90,2] + 15.038;
   1:L PR[91] R[100]mm/sec CNT100;
   1:  PR[GP1:91,1] = PR[GP1:90,1] + -30.823;
   1:  PR[GP1:91,2] = PR[GP1:90,2] + 14.146;
   1:L PR[91] R[100]mm/sec CNT100;
   1:  PR[GP1:91,1] = PR[GP1:90,1] + -32.542;
   1:  PR[GP1:91,2] = PR[GP1:90,2] + 12.290;
   1:L PR[91] R[100]mm/sec CNT100;
   1:  PR[GP1:91,1] = PR[GP1:90,1] + -33.292;
   1:  PR[GP1:91,2] = PR[GP1:90,2] + 11.357;
   1:L PR[91] R[100]mm/sec CNT100;
   1:  PR[GP1:91,1] = PR[GP1:90,1] + -34.740;
   1:  PR[GP1:91,2] = PR[GP1:90,2] + 9.157;
   1:L PR[91] R[100]mm/sec CNT100;
   1:  PR[GP1:91,1] = PR[GP1:90,1] + -36.271;
   1:  PR[GP1:91,2] = PR[GP1:90,2] + 5.723;
   1:L PR[91] R[100]mm/sec CNT100;
   1:  PR[GP1:91,1] = PR[GP1:90,1] + -36.927;
   1:  PR[GP1:91,2] = PR[GP1:90,2] + 3.192;
   1:L PR[91] R[100]mm/sec CNT100;
   1:  PR[GP1:91,1] = PR[GP1:90,1] + -37.152;
   1:  PR[GP1:91,2] = PR[GP1:90,2] + 0.370;
   1:L PR[91] R[100]mm/sec CNT100;
   1:  PR[GP1:91,1] = PR[GP1:90,1] + -37.253;
   1:  PR[GP1:91,2] = PR[GP1:90,2] + -0.354;
   1:L PR[91] R[100]mm/sec CNT100;
   1:  PR[GP1:91,1] = PR[GP1:90,1] + -37.039;
   1:  PR[GP1:91,2] = PR[GP1:90,2] + -3.046;
   1:L PR[91] R[100]mm/sec CNT100;
   1:  PR[GP1:91,1] = PR[GP1:90,1] + -36.937;
   1:  PR[GP1:91,2] = PR[GP1:90,2] + -3.776;
   1:L PR[91] R[100]mm/sec CNT100;
   1:  PR[GP1:91,1] = PR[GP1:90,1] + -36.272;
   1:  PR[GP1:91,2] = PR[GP1:90,2] + -6.346;
   1:L PR[91] R[100]mm/sec CNT100;
   1:  PR[GP1:91,1] = PR[GP1:90,1] + -35.123;
   1:  PR[GP1:91,2] = PR[GP1:90,2] + -8.906;
   1:L PR[91] R[100]mm/sec CNT100;
   1:  PR[GP1:91,1] = PR[GP1:90,1] + -34.737;
   1:  PR[GP1:91,2] = PR[GP1:90,2] + -9.787;
   1:L PR[91] R[100]mm/sec CNT100;
   1:  PR[GP1:91,1] = PR[GP1:90,1] + -33.291;
   1:  PR[GP1:91,2] = PR[GP1:90,2] + -11.984;
   1:L PR[91] R[100]mm/sec CNT100;
   1:  PR[GP1:91,1] = PR[GP1:90,1] + -32.538;
   1:  PR[GP1:91,2] = PR[GP1:90,2] + -12.917;
   1:L PR[91] R[100]mm/sec CNT100;
   1:  PR[GP1:91,1] = PR[GP1:90,1] + -30.802;
   1:  PR[GP1:91,2] = PR[GP1:90,2] + -14.793;
   1:L PR[91] R[100]mm/sec CNT100;
   1:  PR[GP1:91,1] = PR[GP1:90,1] + -28.914;
   1:  PR[GP1:91,2] = PR[GP1:90,2] + -16.270;
   1:L PR[91] R[100]mm/sec CNT100;
   1:  PR[GP1:91,1] = PR[GP1:90,1] + -27.550;
   1:  PR[GP1:91,2] = PR[GP1:90,2] + -17.259;
   1:L PR[91] R[100]mm/sec CNT100;
   1:  PR[GP1:91,1] = PR[GP1:90,1] + -25.557;
   1:  PR[GP1:91,2] = PR[GP1:90,2] + -18.375;
   1:L PR[91] R[100]mm/sec CNT100;
   1:  PR[GP1:91,1] = PR[GP1:90,1] + -23.556;
   1:  PR[GP1:91,2] = PR[GP1:90,2] + -19.114;
   1:L PR[91] R[100]mm/sec CNT100;
   1:  PR[GP1:91,1] = PR[GP1:90,1] + -21.478;
   1:  PR[GP1:91,2] = PR[GP1:90,2] + -19.925;
   1:L PR[91] R[100]mm/sec CNT100;
   1:  PR[GP1:91,1] = PR[GP1:90,1] + -19.584;
   1:  PR[GP1:91,2] = PR[GP1:90,2] + -20.318;
   1:L PR[91] R[100]mm/sec CNT100;
   1:  PR[GP1:91,1] = PR[GP1:90,1] + -16.934;
   1:  PR[GP1:91,2] = PR[GP1:90,2] + -20.626;
   1:L PR[91] R[100]mm/sec CNT100;
   1:  PR[GP1:91,1] = PR[GP1:90,1] + -15.108;
   1:  PR[GP1:91,2] = PR[GP1:90,2] + -20.723;
   1:L PR[91] R[100]mm/sec CNT100;
   1:  PR[GP1:91,1] = PR[GP1:90,1] + -13.486;
   1:  PR[GP1:91,2] = PR[GP1:90,2] + -20.559;
   1:L PR[91] R[100]mm/sec CNT100;
   1:  PR[GP1:91,1] = PR[GP1:90,1] + -10.336;
   1:  PR[GP1:91,2] = PR[GP1:90,2] + -20.119;
   1:L PR[91] R[100]mm/sec CNT100;
   1:  PR[GP1:91,1] = PR[GP1:90,1] + -8.958;
   1:  PR[GP1:91,2] = PR[GP1:90,2] + -19.762;
   1:L PR[91] R[100]mm/sec CNT100;
   1:  PR[GP1:91,1] = PR[GP1:90,1] + -7.715;
   1:  PR[GP1:91,2] = PR[GP1:90,2] + -19.217;
   1:L PR[91] R[100]mm/sec CNT100;
   1:  PR[GP1:91,1] = PR[GP1:90,1] + -4.316;
   1:  PR[GP1:91,2] = PR[GP1:90,2] + -17.769;
   1:L PR[91] R[100]mm/sec CNT100;
   1:  PR[GP1:91,1] = PR[GP1:90,1] + -3.388;
   1:  PR[GP1:91,2] = PR[GP1:90,2] + -17.175;
   1:L PR[91] R[100]mm/sec CNT100;
   1:  PR[GP1:91,1] = PR[GP1:90,1] + -2.398;
   1:  PR[GP1:91,2] = PR[GP1:90,2] + -16.462;
   1:L PR[91] R[100]mm/sec CNT100;
   1:  PR[GP1:91,1] = PR[GP1:90,1] + -1.670;
   1:  PR[GP1:91,2] = PR[GP1:90,2] + -15.824;
   1:L PR[91] R[100]mm/sec CNT100;
   1:  PR[GP1:91,1] = PR[GP1:90,1] + -0.149;
   1:  PR[GP1:91,2] = PR[GP1:90,2] + -15.297;
   1:L PR[91] R[100]mm/sec CNT100;
   1:  PR[GP1:91,1] = PR[GP1:90,1] + 1.655;
   1:  PR[GP1:91,2] = PR[GP1:90,2] + -15.626;
   1:L PR[91] R[100]mm/sec CNT100;
   1:  PR[GP1:91,1] = PR[GP1:90,1] + 1.896;
   1:  PR[GP1:91,2] = PR[GP1:90,2] + -15.900;
   1:L PR[91] R[100]mm/sec CNT100;
   1:  PR[GP1:91,1] = PR[GP1:90,1] + 1.942;
   1:  PR[GP1:91,2] = PR[GP1:90,2] + -15.927;
   1:L PR[91] R[100]mm/sec CNT100;
   1:  PR[GP1:91,1] = PR[GP1:90,1] + 2.525;
   1:  PR[GP1:91,2] = PR[GP1:90,2] + -16.439;
   1:L PR[91] R[100]mm/sec CNT100;
   1:  PR[GP1:91,1] = PR[GP1:90,1] + 2.844;
   1:  PR[GP1:91,2] = PR[GP1:90,2] + -16.643;
   1:L PR[91] R[100]mm/sec CNT100;
   1:  PR[GP1:91,1] = PR[GP1:90,1] + 3.511;
   1:  PR[GP1:91,2] = PR[GP1:90,2] + -17.118;
   1:L PR[91] R[100]mm/sec CNT100;
   1:  PR[GP1:91,1] = PR[GP1:90,1] + 4.486;
   1:  PR[GP1:91,2] = PR[GP1:90,2] + -17.777;
   1:L PR[91] R[100]mm/sec CNT100;
   1:  PR[GP1:91,1] = PR[GP1:90,1] + 9.104;
   1:  PR[GP1:91,2] = PR[GP1:90,2] + -19.757;
   1:L PR[91] R[100]mm/sec CNT100;
   1:  PR[GP1:91,1] = PR[GP1:90,1] + 10.466;
   1:  PR[GP1:91,2] = PR[GP1:90,2] + -20.110;
   1:L PR[91] R[100]mm/sec CNT100;
   1:  PR[GP1:91,1] = PR[GP1:90,1] + 12.188;
   1:  PR[GP1:91,2] = PR[GP1:90,2] + -20.291;
   1:L PR[91] R[100]mm/sec CNT100;
   1:  PR[GP1:91,1] = PR[GP1:90,1] + 15.286;
   1:  PR[GP1:91,2] = PR[GP1:90,2] + -20.722;
   1:L PR[91] R[100]mm/sec CNT100;
   1:  PR[GP1:91,1] = PR[GP1:90,1] + 17.075;
   1:  PR[GP1:91,2] = PR[GP1:90,2] + -20.629;
   1:L PR[91] R[100]mm/sec CNT100;
   1:  PR[GP1:91,1] = PR[GP1:90,1] + 19.726;
   1:  PR[GP1:91,2] = PR[GP1:90,2] + -20.320;
   1:L PR[91] R[100]mm/sec CNT100;
   1:  PR[GP1:91,1] = PR[GP1:90,1] + 21.629;
   1:  PR[GP1:91,2] = PR[GP1:90,2] + -19.926;
   1:L PR[91] R[100]mm/sec CNT100;
   1:  PR[GP1:91,1] = PR[GP1:90,1] + 23.740;
   1:  PR[GP1:91,2] = PR[GP1:90,2] + -19.146;
   1:L PR[91] R[100]mm/sec CNT100;
   1:  PR[GP1:91,1] = PR[GP1:90,1] + 25.690;
   1:  PR[GP1:91,2] = PR[GP1:90,2] + -18.388;
   1:L PR[91] R[100]mm/sec CNT100;
   1:  PR[GP1:91,1] = PR[GP1:90,1] + 27.664;
   1:  PR[GP1:91,2] = PR[GP1:90,2] + -17.288;
   1:L PR[91] R[100]mm/sec CNT100;
   1:  PR[GP1:91,1] = PR[GP1:90,1] + 29.708;
   1:  PR[GP1:91,2] = PR[GP1:90,2] + -15.704;
   1:L PR[91] R[100]mm/sec CNT100;
   1:  PR[GP1:91,1] = PR[GP1:90,1] + 30.938;
   1:  PR[GP1:91,2] = PR[GP1:90,2] + -14.810;
   1:L PR[91] R[100]mm/sec CNT100;
   1:  PR[GP1:91,1] = PR[GP1:90,1] + 32.661;
   1:  PR[GP1:91,2] = PR[GP1:90,2] + -12.952;
   1:L PR[91] R[100]mm/sec CNT100;
   1:  PR[GP1:91,1] = PR[GP1:90,1] + 33.417;
   1:  PR[GP1:91,2] = PR[GP1:90,2] + -12.013;
   1:L PR[91] R[100]mm/sec CNT100;
   1:  PR[GP1:91,1] = PR[GP1:90,1] + 34.886;
   1:  PR[GP1:91,2] = PR[GP1:90,2] + -9.794;
   1:L PR[91] R[100]mm/sec CNT100;
   1:  PR[GP1:91,1] = PR[GP1:90,1] + 36.073;
   1:  PR[GP1:91,2] = PR[GP1:90,2] + -7.179;
   1:L PR[91] R[100]mm/sec CNT100;
   1:  PR[GP1:91,1] = PR[GP1:90,1] + 36.413;
   1:  PR[GP1:91,2] = PR[GP1:90,2] + -6.408;
   1:L PR[91] R[100]mm/sec CNT100;
   1:  PR[GP1:91,1] = PR[GP1:90,1] + 37.071;
   1:  PR[GP1:91,2] = PR[GP1:90,2] + -3.903;
   1:L PR[91] R[100]mm/sec CNT100;
   1:  PR[GP1:91,1] = PR[GP1:90,1] + 37.309;
   1:  PR[GP1:91,2] = PR[GP1:90,2] + -0.996;
   1:L PR[91] R[100]mm/sec CNT100;
   1:  PR[GP1:91,1] = PR[GP1:90,1] + 37.409;
   1:  PR[GP1:91,2] = PR[GP1:90,2] + -0.271;
   1:L PR[91] R[100]mm/sec CNT100;
   1:  PR[GP1:91,1] = PR[GP1:90,1] + 37.183;
   1:  PR[GP1:91,2] = PR[GP1:90,2] + 2.507;
   1:L PR[91] R[100]mm/sec CNT100;
   1:  PR[GP1:91,1] = PR[GP1:90,1] + 37.081;
   1:  PR[GP1:91,2] = PR[GP1:90,2] + 3.239;
   1:L PR[91] R[100]mm/sec CNT100;
   1:  PR[GP1:91,1] = PR[GP1:90,1] + 36.415;
   1:  PR[GP1:91,2] = PR[GP1:90,2] + 5.777;
   1:L PR[91] R[100]mm/sec CNT100;
   1:  PR[GP1:91,1] = PR[GP1:90,1] + 34.887;
   1:  PR[GP1:91,2] = PR[GP1:90,2] + 9.169;
   1:L PR[91] R[100]mm/sec CNT100;
   1:  PR[GP1:91,1] = PR[GP1:90,1] + 33.418;
   1:  PR[GP1:91,2] = PR[GP1:90,2] + 11.387;
   1:L PR[91] R[100]mm/sec CNT100;
   1:  PR[GP1:91,1] = PR[GP1:90,1] + 32.665;
   1:  PR[GP1:91,2] = PR[GP1:90,2] + 12.325;
   1:L PR[91] R[100]mm/sec CNT100;
   1:  PR[GP1:91,1] = PR[GP1:90,1] + 30.926;
   1:  PR[GP1:91,2] = PR[GP1:90,2] + 14.200;
   1:L PR[91] R[100]mm/sec CNT100;
   1:  PR[GP1:91,1] = PR[GP1:90,1] + 29.053;
   1:  PR[GP1:91,2] = PR[GP1:90,2] + 15.659;
   1:L PR[91] R[100]mm/sec CNT100;
   1:  PR[GP1:91,1] = PR[GP1:90,1] + 27.692;
   1:  PR[GP1:91,2] = PR[GP1:90,2] + 16.648;
   1:L PR[91] R[100]mm/sec CNT100;
   1:  PR[GP1:91,1] = PR[GP1:90,1] + 25.711;
   1:  PR[GP1:91,2] = PR[GP1:90,2] + 17.752;
   1:L PR[91] R[100]mm/sec CNT100;
   1:  PR[GP1:91,1] = PR[GP1:90,1] + 23.706;
   1:  PR[GP1:91,2] = PR[GP1:90,2] + 18.489;
   1:L PR[91] R[100]mm/sec CNT100;
   1:  PR[GP1:91,1] = PR[GP1:90,1] + 21.631;
   1:  PR[GP1:91,2] = PR[GP1:90,2] + 19.301;
   1:L PR[91] R[100]mm/sec CNT100;
   1:  PR[GP1:91,1] = PR[GP1:90,1] + 19.740;
   1:  PR[GP1:91,2] = PR[GP1:90,2] + 19.692;
   1:L PR[91] R[100]mm/sec CNT100;
   1:  PR[GP1:91,1] = PR[GP1:90,1] + 17.096;
   1:  PR[GP1:91,2] = PR[GP1:90,2] + 20.005;
   1:L PR[91] R[100]mm/sec CNT100;
   1:  PR[GP1:91,1] = PR[GP1:90,1] + 15.281;
   1:  PR[GP1:91,2] = PR[GP1:90,2] + 20.099;
   1:L PR[91] R[100]mm/sec CNT100;
   1:  PR[GP1:91,1] = PR[GP1:90,1] + 13.662;
   1:  PR[GP1:91,2] = PR[GP1:90,2] + 19.935;
   1:L PR[91] R[100]mm/sec CNT100;
   1:  PR[GP1:91,1] = PR[GP1:90,1] + 10.518;
   1:  PR[GP1:91,2] = PR[GP1:90,2] + 19.500;
   1:L PR[91] R[100]mm/sec CNT100;
   1:  PR[GP1:91,1] = PR[GP1:90,1] + 9.138;
   1:  PR[GP1:91,2] = PR[GP1:90,2] + 19.142;
   1:L PR[91] R[100]mm/sec CNT100;
   1:  PR[GP1:91,1] = PR[GP1:90,1] + 7.893;
   1:  PR[GP1:91,2] = PR[GP1:90,2] + 18.598;
   1:L PR[91] R[100]mm/sec CNT100;
   1:  PR[GP1:91,1] = PR[GP1:90,1] + 4.564;
   1:  PR[GP1:91,2] = PR[GP1:90,2] + 17.206;
   1:L PR[91] R[100]mm/sec CNT100;
   1:  PR[GP1:91,1] = PR[GP1:90,1] + 3.599;
   1:  PR[GP1:91,2] = PR[GP1:90,2] + 16.590;
   1:L PR[91] R[100]mm/sec CNT100;
   1:  PR[GP1:91,1] = PR[GP1:90,1] + 2.963;
   1:  PR[GP1:91,2] = PR[GP1:90,2] + 16.151;
   1:L PR[91] R[100]mm/sec CNT100;
   1:  PR[GP1:91,1] = PR[GP1:90,1] + 2.037;
   1:  PR[GP1:91,2] = PR[GP1:90,2] + 15.418;
   1:L PR[91] R[100]mm/sec CNT100;
   1:  PR[GP1:91,1] = PR[GP1:90,1] + 1.582;
   1:  PR[GP1:91,2] = PR[GP1:90,2] + 14.977;
   1:L PR[91] R[100]mm/sec CNT100;
   1:  PR[GP1:91,1] = PR[GP1:90,1] + -0.181;
   1:  PR[GP1:91,2] = PR[GP1:90,2] + 14.671;
   1:L PR[91] R[100]mm/sec CNT100;
   1:  PR[91] = PR[90];
   1:  PR[GP1:91,1] = PR[GP1:90,1] + -1.636;
   1:  PR[GP1:91,2] = PR[GP1:90,2] + 15.480;
   1:  PR[GP1:91,3] = PR[GP1:90,3] + 34.465;
   1:L PR[91] R[100]mm/sec CNT100;
   1:  PR[GP1:91,1] = PR[GP1:90,1] + -2.573;
   1:  PR[GP1:91,2] = PR[GP1:90,2] + 16.221;
   1:L PR[91] R[100]mm/sec CNT100;
   1:  PR[GP1:91,1] = PR[GP1:90,1] + -4.144;
   1:  PR[GP1:91,2] = PR[GP1:90,2] + 17.260;
   1:L PR[91] R[100]mm/sec CNT100;
   1:  PR[GP1:91,1] = PR[GP1:90,1] + -5.225;
   1:  PR[GP1:91,2] = PR[GP1:90,2] + 17.732;
   1:L PR[91] R[100]mm/sec CNT100;
   1:  PR[GP1:91,1] = PR[GP1:90,1] + -8.781;
   1:  PR[GP1:91,2] = PR[GP1:90,2] + 19.222;
   1:L PR[91] R[100]mm/sec CNT100;
   1:  PR[GP1:91,1] = PR[GP1:90,1] + -10.016;
   1:  PR[GP1:91,2] = PR[GP1:90,2] + 19.542;
   1:L PR[91] R[100]mm/sec CNT100;
   1:  PR[GP1:91,1] = PR[GP1:90,1] + -11.593;
   1:  PR[GP1:91,2] = PR[GP1:90,2] + 19.706;
   1:L PR[91] R[100]mm/sec CNT100;
   1:  PR[GP1:91,1] = PR[GP1:90,1] + -14.933;
   1:  PR[GP1:91,2] = PR[GP1:90,2] + 20.162;
   1:L PR[91] R[100]mm/sec CNT100;
   1:  PR[GP1:91,1] = PR[GP1:90,1] + -16.588;
   1:  PR[GP1:91,2] = PR[GP1:90,2] + 20.074;
   1:L PR[91] R[100]mm/sec CNT100;
   1:  PR[GP1:91,1] = PR[GP1:90,1] + -19.474;
   1:  PR[GP1:91,2] = PR[GP1:90,2] + 19.733;
   1:L PR[91] R[100]mm/sec CNT100;
   1:  PR[GP1:91,1] = PR[GP1:90,1] + -21.247;
   1:  PR[GP1:91,2] = PR[GP1:90,2] + 19.365;
   1:L PR[91] R[100]mm/sec CNT100;
   1:  PR[GP1:91,1] = PR[GP1:90,1] + -23.211;
   1:  PR[GP1:91,2] = PR[GP1:90,2] + 18.636;
   1:L PR[91] R[100]mm/sec CNT100;
   1:  PR[GP1:91,1] = PR[GP1:90,1] + -25.393;
   1:  PR[GP1:91,2] = PR[GP1:90,2] + 17.783;
   1:L PR[91] R[100]mm/sec CNT100;
   1:  PR[GP1:91,1] = PR[GP1:90,1] + -27.250;
   1:  PR[GP1:91,2] = PR[GP1:90,2] + 16.743;
   1:L PR[91] R[100]mm/sec CNT100;
   1:  PR[GP1:91,1] = PR[GP1:90,1] + -29.186;
   1:  PR[GP1:91,2] = PR[GP1:90,2] + 15.236;
   1:L PR[91] R[100]mm/sec CNT100;
   1:  PR[GP1:91,1] = PR[GP1:90,1] + -30.627;
   1:  PR[GP1:91,2] = PR[GP1:90,2] + 14.187;
   1:L PR[91] R[100]mm/sec CNT100;
   1:  PR[GP1:91,1] = PR[GP1:90,1] + -32.246;
   1:  PR[GP1:91,2] = PR[GP1:90,2] + 12.438;
   1:L PR[91] R[100]mm/sec CNT100;
   1:  PR[GP1:91,1] = PR[GP1:90,1] + -33.157;
   1:  PR[GP1:91,2] = PR[GP1:90,2] + 11.306;
   1:L PR[91] R[100]mm/sec CNT100;
   1:  PR[GP1:91,1] = PR[GP1:90,1] + -34.525;
   1:  PR[GP1:91,2] = PR[GP1:90,2] + 9.226;
   1:L PR[91] R[100]mm/sec CNT100;
   1:  PR[GP1:91,1] = PR[GP1:90,1] + -36.097;
   1:  PR[GP1:91,2] = PR[GP1:90,2] + 5.698;
   1:L PR[91] R[100]mm/sec CNT100;
   1:  PR[GP1:91,1] = PR[GP1:90,1] + -36.716;
   1:  PR[GP1:91,2] = PR[GP1:90,2] + 3.304;
   1:L PR[91] R[100]mm/sec CNT100;
   1:  PR[GP1:91,1] = PR[GP1:90,1] + -36.931;
   1:  PR[GP1:91,2] = PR[GP1:90,2] + 0.625;
   1:L PR[91] R[100]mm/sec CNT100;
   1:  PR[GP1:91,1] = PR[GP1:90,1] + -37.067;
   1:  PR[GP1:91,2] = PR[GP1:90,2] + -0.354;
   1:L PR[91] R[100]mm/sec CNT100;
   1:  PR[GP1:91,1] = PR[GP1:90,1] + -36.864;
   1:  PR[GP1:91,2] = PR[GP1:90,2] + -2.907;
   1:L PR[91] R[100]mm/sec CNT100;
   1:  PR[GP1:91,1] = PR[GP1:90,1] + -36.727;
   1:  PR[GP1:91,2] = PR[GP1:90,2] + -3.888;
   1:L PR[91] R[100]mm/sec CNT100;
   1:  PR[GP1:91,1] = PR[GP1:90,1] + -36.097;
   1:  PR[GP1:91,2] = PR[GP1:90,2] + -6.321;
   1:L PR[91] R[100]mm/sec CNT100;
   1:  PR[GP1:91,1] = PR[GP1:90,1] + -35.007;
   1:  PR[GP1:91,2] = PR[GP1:90,2] + -8.749;
   1:L PR[91] R[100]mm/sec CNT100;
   1:  PR[GP1:91,1] = PR[GP1:90,1] + -34.521;
   1:  PR[GP1:91,2] = PR[GP1:90,2] + -9.857;
   1:L PR[91] R[100]mm/sec CNT100;
   1:  PR[GP1:91,1] = PR[GP1:90,1] + -33.155;
   1:  PR[GP1:91,2] = PR[GP1:90,2] + -11.933;
   1:L PR[91] R[100]mm/sec CNT100;
   1:  PR[GP1:91,1] = PR[GP1:90,1] + -32.242;
   1:  PR[GP1:91,2] = PR[GP1:90,2] + -13.065;
   1:L PR[91] R[100]mm/sec CNT100;
   1:  PR[GP1:91,1] = PR[GP1:90,1] + -30.605;
   1:  PR[GP1:91,2] = PR[GP1:90,2] + -14.834;
   1:L PR[91] R[100]mm/sec CNT100;
   1:  PR[GP1:91,1] = PR[GP1:90,1] + -28.825;
   1:  PR[GP1:91,2] = PR[GP1:90,2] + -16.227;
   1:L PR[91] R[100]mm/sec CNT100;
   1:  PR[GP1:91,1] = PR[GP1:90,1] + -27.261;
   1:  PR[GP1:91,2] = PR[GP1:90,2] + -17.360;
   1:L PR[91] R[100]mm/sec CNT100;
   1:  PR[GP1:91,1] = PR[GP1:90,1] + -25.395;
   1:  PR[GP1:91,2] = PR[GP1:90,2] + -18.406;
   1:L PR[91] R[100]mm/sec CNT100;
   1:  PR[GP1:91,1] = PR[GP1:90,1] + -23.516;
   1:  PR[GP1:91,2] = PR[GP1:90,2] + -19.100;
   1:L PR[91] R[100]mm/sec CNT100;
   1:  PR[GP1:91,1] = PR[GP1:90,1] + -21.218;
   1:  PR[GP1:91,2] = PR[GP1:90,2] + -19.996;
   1:L PR[91] R[100]mm/sec CNT100;
   1:  PR[GP1:91,1] = PR[GP1:90,1] + -19.458;
   1:  PR[GP1:91,2] = PR[GP1:90,2] + -20.361;
   1:L PR[91] R[100]mm/sec CNT100;
   1:  PR[GP1:91,1] = PR[GP1:90,1] + -16.565;
   1:  PR[GP1:91,2] = PR[GP1:90,2] + -20.698;
   1:L PR[91] R[100]mm/sec CNT100;
   1:  PR[GP1:91,1] = PR[GP1:90,1] + -14.882;
   1:  PR[GP1:91,2] = PR[GP1:90,2] + -20.787;
   1:L PR[91] R[100]mm/sec CNT100;
   1:  PR[GP1:91,1] = PR[GP1:90,1] + -13.387;
   1:  PR[GP1:91,2] = PR[GP1:90,2] + -20.636;
   1:L PR[91] R[100]mm/sec CNT100;
   1:  PR[GP1:91,1] = PR[GP1:90,1] + -10.009;
   1:  PR[GP1:91,2] = PR[GP1:90,2] + -20.163;
   1:L PR[91] R[100]mm/sec CNT100;
   1:  PR[GP1:91,1] = PR[GP1:90,1] + -8.760;
   1:  PR[GP1:91,2] = PR[GP1:90,2] + -19.840;
   1:L PR[91] R[100]mm/sec CNT100;
   1:  PR[GP1:91,1] = PR[GP1:90,1] + -7.628;
   1:  PR[GP1:91,2] = PR[GP1:90,2] + -19.344;
   1:L PR[91] R[100]mm/sec CNT100;
   1:  PR[GP1:91,1] = PR[GP1:90,1] + -4.022;
   1:  PR[GP1:91,2] = PR[GP1:90,2] + -17.808;
   1:L PR[91] R[100]mm/sec CNT100;
   1:  PR[GP1:91,1] = PR[GP1:90,1] + -3.202;
   1:  PR[GP1:91,2] = PR[GP1:90,2] + -17.283;
   1:L PR[91] R[100]mm/sec CNT100;
   1:  PR[GP1:91,1] = PR[GP1:90,1] + -2.154;
   1:  PR[GP1:91,2] = PR[GP1:90,2] + -16.528;
   1:L PR[91] R[100]mm/sec CNT100;
   1:  PR[GP1:91,1] = PR[GP1:90,1] + -1.649;
   1:  PR[GP1:91,2] = PR[GP1:90,2] + -16.085;
   1:L PR[91] R[100]mm/sec CNT100;
   1:  PR[GP1:91,1] = PR[GP1:90,1] + -0.861;
   1:  PR[GP1:91,2] = PR[GP1:90,2] + -15.817;
   1:L PR[91] R[100]mm/sec CNT100;
   1:  PR[GP1:91,1] = PR[GP1:90,1] + -0.023;
   1:  PR[GP1:91,2] = PR[GP1:90,2] + -15.471;
   1:L PR[91] R[100]mm/sec CNT100;
   1:  PR[GP1:91,1] = PR[GP1:90,1] + 0.569;
   1:  PR[GP1:91,2] = PR[GP1:90,2] + -15.707;
   1:L PR[91] R[100]mm/sec CNT100;
   1:  PR[GP1:91,1] = PR[GP1:90,1] + 1.674;
   1:  PR[GP1:91,2] = PR[GP1:90,2] + -15.905;
   1:L PR[91] R[100]mm/sec CNT100;
   1:  PR[GP1:91,1] = PR[GP1:90,1] + 1.933;
   1:  PR[GP1:91,2] = PR[GP1:90,2] + -16.199;
   1:L PR[91] R[100]mm/sec CNT100;
   1:  PR[GP1:91,1] = PR[GP1:90,1] + 2.296;
   1:  PR[GP1:91,2] = PR[GP1:90,2] + -16.518;
   1:L PR[91] R[100]mm/sec CNT100;
   1:  PR[GP1:91,1] = PR[GP1:90,1] + 4.197;
   1:  PR[GP1:91,2] = PR[GP1:90,2] + -17.817;
   1:L PR[91] R[100]mm/sec CNT100;
   1:  PR[GP1:91,1] = PR[GP1:90,1] + 8.906;
   1:  PR[GP1:91,2] = PR[GP1:90,2] + -19.835;
   1:L PR[91] R[100]mm/sec CNT100;
   1:  PR[GP1:91,1] = PR[GP1:90,1] + 10.139;
   1:  PR[GP1:91,2] = PR[GP1:90,2] + -20.155;
   1:L PR[91] R[100]mm/sec CNT100;
   1:  PR[GP1:91,1] = PR[GP1:90,1] + 11.713;
   1:  PR[GP1:91,2] = PR[GP1:90,2] + -20.320;
   1:L PR[91] R[100]mm/sec CNT100;
   1:  PR[GP1:91,1] = PR[GP1:90,1] + 15.060;
   1:  PR[GP1:91,2] = PR[GP1:90,2] + -20.786;
   1:L PR[91] R[100]mm/sec CNT100;
   1:  PR[GP1:91,1] = PR[GP1:90,1] + 16.707;
   1:  PR[GP1:91,2] = PR[GP1:90,2] + -20.700;
   1:L PR[91] R[100]mm/sec CNT100;
   1:  PR[GP1:91,1] = PR[GP1:90,1] + 19.600;
   1:  PR[GP1:91,2] = PR[GP1:90,2] + -20.363;
   1:L PR[91] R[100]mm/sec CNT100;
   1:  PR[GP1:91,1] = PR[GP1:90,1] + 21.371;
   1:  PR[GP1:91,2] = PR[GP1:90,2] + -19.996;
   1:L PR[91] R[100]mm/sec CNT100;
   1:  PR[GP1:91,1] = PR[GP1:90,1] + 23.338;
   1:  PR[GP1:91,2] = PR[GP1:90,2] + -19.270;
   1:L PR[91] R[100]mm/sec CNT100;
   1:  PR[GP1:91,1] = PR[GP1:90,1] + 25.528;
   1:  PR[GP1:91,2] = PR[GP1:90,2] + -18.418;
   1:L PR[91] R[100]mm/sec CNT100;
   1:  PR[GP1:91,1] = PR[GP1:90,1] + 27.377;
   1:  PR[GP1:91,2] = PR[GP1:90,2] + -17.388;
   1:L PR[91] R[100]mm/sec CNT100;
   1:  PR[GP1:91,1] = PR[GP1:90,1] + 29.297;
   1:  PR[GP1:91,2] = PR[GP1:90,2] + -15.900;
   1:L PR[91] R[100]mm/sec CNT100;
   1:  PR[GP1:91,1] = PR[GP1:90,1] + 30.743;
   1:  PR[GP1:91,2] = PR[GP1:90,2] + -14.849;
   1:L PR[91] R[100]mm/sec CNT100;
   1:  PR[GP1:91,1] = PR[GP1:90,1] + 32.366;
   1:  PR[GP1:91,2] = PR[GP1:90,2] + -13.099;
   1:L PR[91] R[100]mm/sec CNT100;
   1:  PR[GP1:91,1] = PR[GP1:90,1] + 33.283;
   1:  PR[GP1:91,2] = PR[GP1:90,2] + -11.961;
   1:L PR[91] R[100]mm/sec CNT100;
   1:  PR[GP1:91,1] = PR[GP1:90,1] + 34.672;
   1:  PR[GP1:91,2] = PR[GP1:90,2] + -9.862;
   1:L PR[91] R[100]mm/sec CNT100;
   1:  PR[GP1:91,1] = PR[GP1:90,1] + 35.795;
   1:  PR[GP1:91,2] = PR[GP1:90,2] + -7.387;
   1:L PR[91] R[100]mm/sec CNT100;
   1:  PR[GP1:91,1] = PR[GP1:90,1] + 36.239;
   1:  PR[GP1:91,2] = PR[GP1:90,2] + -6.381;
   1:L PR[91] R[100]mm/sec CNT100;
   1:  PR[GP1:91,1] = PR[GP1:90,1] + 36.861;
   1:  PR[GP1:91,2] = PR[GP1:90,2] + -4.011;
   1:L PR[91] R[100]mm/sec CNT100;
   1:  PR[GP1:91,1] = PR[GP1:90,1] + 37.087;
   1:  PR[GP1:91,2] = PR[GP1:90,2] + -1.252;
   1:L PR[91] R[100]mm/sec CNT100;
   1:  PR[GP1:91,1] = PR[GP1:90,1] + 37.223;
   1:  PR[GP1:91,2] = PR[GP1:90,2] + -0.271;
   1:L PR[91] R[100]mm/sec CNT100;
   1:  PR[GP1:91,1] = PR[GP1:90,1] + 37.008;
   1:  PR[GP1:91,2] = PR[GP1:90,2] + 2.364;
   1:L PR[91] R[100]mm/sec CNT100;
   1:  PR[GP1:91,1] = PR[GP1:90,1] + 36.872;
   1:  PR[GP1:91,2] = PR[GP1:90,2] + 3.347;
   1:L PR[91] R[100]mm/sec CNT100;
   1:  PR[GP1:91,1] = PR[GP1:90,1] + 36.242;
   1:  PR[GP1:91,2] = PR[GP1:90,2] + 5.747;
   1:L PR[91] R[100]mm/sec CNT100;
   1:  PR[GP1:91,1] = PR[GP1:90,1] + 35.154;
   1:  PR[GP1:91,2] = PR[GP1:90,2] + 8.139;
   1:L PR[91] R[100]mm/sec CNT100;
   1:  PR[GP1:91,1] = PR[GP1:90,1] + 34.669;
   1:  PR[GP1:91,2] = PR[GP1:90,2] + 9.242;
   1:L PR[91] R[100]mm/sec CNT100;
   1:  PR[GP1:91,1] = PR[GP1:90,1] + 33.284;
   1:  PR[GP1:91,2] = PR[GP1:90,2] + 11.334;
   1:L PR[91] R[100]mm/sec CNT100;
   1:  PR[GP1:91,1] = PR[GP1:90,1] + 32.371;
   1:  PR[GP1:91,2] = PR[GP1:90,2] + 12.471;
   1:L PR[91] R[100]mm/sec CNT100;
   1:  PR[GP1:91,1] = PR[GP1:90,1] + 30.732;
   1:  PR[GP1:91,2] = PR[GP1:90,2] + 14.239;
   1:L PR[91] R[100]mm/sec CNT100;
   1:  PR[GP1:91,1] = PR[GP1:90,1] + 28.966;
   1:  PR[GP1:91,2] = PR[GP1:90,2] + 15.614;
   1:L PR[91] R[100]mm/sec CNT100;
   1:  PR[GP1:91,1] = PR[GP1:90,1] + 27.406;
   1:  PR[GP1:91,2] = PR[GP1:90,2] + 16.748;
   1:L PR[91] R[100]mm/sec CNT100;
   1:  PR[GP1:91,1] = PR[GP1:90,1] + 25.550;
   1:  PR[GP1:91,2] = PR[GP1:90,2] + 17.782;
   1:L PR[91] R[100]mm/sec CNT100;
   1:  PR[GP1:91,1] = PR[GP1:90,1] + 23.667;
   1:  PR[GP1:91,2] = PR[GP1:90,2] + 18.474;
   1:L PR[91] R[100]mm/sec CNT100;
   1:  PR[GP1:91,1] = PR[GP1:90,1] + 21.374;
   1:  PR[GP1:91,2] = PR[GP1:90,2] + 19.371;
   1:L PR[91] R[100]mm/sec CNT100;
   1:  PR[GP1:91,1] = PR[GP1:90,1] + 19.616;
   1:  PR[GP1:91,2] = PR[GP1:90,2] + 19.735;
   1:L PR[91] R[100]mm/sec CNT100;
   1:  PR[GP1:91,1] = PR[GP1:90,1] + 16.730;
   1:  PR[GP1:91,2] = PR[GP1:90,2] + 20.076;
   1:L PR[91] R[100]mm/sec CNT100;
   1:  PR[GP1:91,1] = PR[GP1:90,1] + 15.057;
   1:  PR[GP1:91,2] = PR[GP1:90,2] + 20.163;
   1:L PR[91] R[100]mm/sec CNT100;
   1:  PR[GP1:91,1] = PR[GP1:90,1] + 13.565;
   1:  PR[GP1:91,2] = PR[GP1:90,2] + 20.012;
   1:L PR[91] R[100]mm/sec CNT100;
   1:  PR[GP1:91,1] = PR[GP1:90,1] + 10.193;
   1:  PR[GP1:91,2] = PR[GP1:90,2] + 19.546;
   1:L PR[91] R[100]mm/sec CNT100;
   1:  PR[GP1:91,1] = PR[GP1:90,1] + 8.943;
   1:  PR[GP1:91,2] = PR[GP1:90,2] + 19.221;
   1:L PR[91] R[100]mm/sec CNT100;
   1:  PR[GP1:91,1] = PR[GP1:90,1] + 7.808;
   1:  PR[GP1:91,2] = PR[GP1:90,2] + 18.725;
   1:L PR[91] R[100]mm/sec CNT100;
   1:  PR[GP1:91,1] = PR[GP1:90,1] + 4.277;
   1:  PR[GP1:91,2] = PR[GP1:90,2] + 17.249;
   1:L PR[91] R[100]mm/sec CNT100;
   1:  PR[GP1:91,1] = PR[GP1:90,1] + 3.417;
   1:  PR[GP1:91,2] = PR[GP1:90,2] + 16.700;
   1:L PR[91] R[100]mm/sec CNT100;
   1:  PR[GP1:91,1] = PR[GP1:90,1] + 2.742;
   1:  PR[GP1:91,2] = PR[GP1:90,2] + 16.234;
   1:L PR[91] R[100]mm/sec CNT100;
   1:  PR[GP1:91,1] = PR[GP1:90,1] + 2.019;
   1:  PR[GP1:91,2] = PR[GP1:90,2] + 15.662;
   1:L PR[91] R[100]mm/sec CNT100;
   1:  PR[GP1:91,1] = PR[GP1:90,1] + 1.599;
   1:  PR[GP1:91,2] = PR[GP1:90,2] + 15.256;
   1:L PR[91] R[100]mm/sec CNT100;
   1:  PR[GP1:91,1] = PR[GP1:90,1] + 0.552;
   1:  PR[GP1:91,2] = PR[GP1:90,2] + 15.077;
   1:L PR[91] R[100]mm/sec CNT100;
   1:  PR[GP1:91,1] = PR[GP1:90,1] + -0.002;
   1:  PR[GP1:91,2] = PR[GP1:90,2] + 14.853;
   1:L PR[91] R[100]mm/sec CNT100 TB   .50sec,CALL END_PUD;
   1:  DO[117:Laser Start]=OFF;
   1:  PR[92] = PR[91];
   1:  PR[GP1:92,3] = PR[GP1:92,3] + 50;
   1:J PR[92] 10% FINE;
   1:  WAIT   5.00(sec);
   1:  DO[119:Gas]=OFF;
   1:  CALL HOME_ALL;
/POS
/END
